// ObjectHandling/GlobalObjects
{attribute 'qualified_only'}
{attribute 'global_init_slot' := '49995'}
VAR_GLOBAL CONSTANT
	MAX_OBJECTS : UINT := 750;
	MAX_CYLINDERS : UINT := 20;
	MAX_MOTORS : UINT := 10;
	MAX_FAULTS : UINT := 300;
	MAX_LOGS : UINT := 100;
	MAX_LOGGABLE : UINT := 500;
	MAX_EXECUTEABLE : UINT := 300;
END_VAR

VAR_GLOBAL
	CollectionOfAllObjects : FB_CollectionHandlerAll; 
	CollectionOfFaults : FB_CollectionHandlerFaults; 
// 	CollectionOfCylinders : FB_CollectionHandlerCylinders;
// 	CollectionOfPositionableMotors : FB_CollectionHandlerPositionableMotors;
	CollectionOfActiveFaults : FB_CollectionHandlerActiveFaults; 
	CollectionOfLogs : FB_CollectionHandlerLogs; 
	CollectionOfLoggable : FB_CollectionHandlerLoggable;
	CollectionOfExecutable : FB_CollectionHandlerExecutable;
	CollectionOfInitialzable : FB_CollectionHandlerInitializable;
	Reversing: INT;
END_VAR

// RemoteComms/RemoteComms
{attribute 'qualified_only'}
VAR_GLOBAL
	OPCInputsToBagger : OPC_Inputs;
	OPCOutputsFromBagger : OPC_Outputs;
	modbusInputsToBagger : Modbus_Inputs;
	modbusOutputsFromBagger : Modbus_Outputs;
END_VAR

// UN00 - Sharp Bagger/UN00_Globals
{attribute 'qualified_only'}
VAR_GLOBAL
	simFaults : FB_Simulation();
END_VAR

VAR_GLOBAL CONSTANT
	sAutomatic : STRING := 'Automatic';
	sSemiAuto : STRING := 'Semi-Auto';
	sMaintenance : STRING := 'Maintenance';
	sSimulation : STRING := 'Simulation';
	
END_VAR

// FBs/FB_CycleCounter
FUNCTION_BLOCK FB_CycleCounter
VAR_INPUT
	reset : BOOL;
END_VAR
VAR_OUTPUT
END_VAR
VAR
    count : UDINT;
END_VAR

IF reset THEN
	THIS^.Clear();
	reset := FALSE;
END_IF

METHOD Clear
VAR_INPUT
END_VAR
count := 0;
END_METHOD

METHOD Increment
VAR_INPUT
END_VAR
count := count + 1;
END_METHOD

METHOD SetCount
VAR_INPUT
	countSetting : UDINT;
END_VAR
count := countSetting;
END_METHOD

END_FUNCTION_BLOCK

// FBs/FB_CylinderLeak
FUNCTION_BLOCK FB_CylinderLeak EXTENDS FB_PredictiveMaint
VAR_INPUT
	iExtended : BOOL;
	iRetracted : BOOL;
	maximumStrokeTime : REAL;
END_VAR
VAR_OUTPUT
	strokeTime : REAL;
END_VAR
VAR
	strokeTimer : TON := (PT := T#1H);
	extendedONS : R_TRIG;
	retractedONS : R_TRIG;
END_VAR

extendedONS(CLK := iExtended);
retractedONS(CLK := iRetracted);

IF extendedONS.Q OR retractedONS.Q THEN
	strokeTime := TO_REAL(strokeTimer.ET) / 1000;
END_IF

strokeTimer(IN := NOT iExtended AND NOT iRetracted);

END_FUNCTION_BLOCK

// FBs/FB_PredictiveMaint
FUNCTION_BLOCK FB_PredictiveMaint EXTENDS FB_CycleCounter
VAR_INPUT
	target : UDINT;
	name : STRING;
	units : STRING := 'Machine Cycles';
END_VAR
VAR_OUTPUT
	
END_VAR
VAR
	
END_VAR

SUPER^();

END_FUNCTION_BLOCK

// FBs/FB_DeviceTreeEnable
{attribute 'analysis' := '-169, -34'}FUNCTION_BLOCK FB_DeviceTreeEnable
VAR_INPUT
	rootEIPNode : DED.INode;
	rootModbusTCPNode : DED.INode;
END_VAR
VAR
	reconfigEIP : DED.Reconfigure;
	reconfigModbusTCP : DED.Reconfigure;
	deviceState : DED.DEVICE_STATE;
	_recongfigCommand : BOOL;
	state : INT;
	disabledSettingWordEIP : DWORD;
	disabledStatusWordEIP : DWORD;
	disabledSettingWordModbusTCP : DWORD;
	disabledStatusWordModbusTCP : DWORD;
END_VAR

VAR_OUTPUT
	
END_VAR

//    Program: FB_EIPCommsConfigure
//    Description: Allows configuration of individual EIP in in the device tree (enable/disable) 
//    For example, to turn off the comms to a Keyence BCV if it isn't installed
//    Created by: Ben Hess
//    Created Date: Wednesday January 6th, 2021

//  Get enable status property
disabledSettingWordEIP.0 := NOT Cube67_BN_E_V2.Enable;
disabledSettingWordEIP.1 := NOT FestoManifold.Enable;
disabledSettingWordEIP.2 := NOT MSFMotor.Enable;
disabledSettingWordEIP.3 := NOT Bag_Delivery_EIP_Motor.Enable;
disabledSettingWordEIP.4 := NOT Bag_Delivery_Rear_Motor.Enable;
disabledSettingWordEIP.5 := NOT Keyence_BCV.Enable;
disabledSettingWordEIP.6 := NOT Infeed_Conveyor_IO.Enable;
disabledSettingWordEIP.7 := NOT Panther_PA.Enable;
disabledSettingWordEIP.8 := NOT IBD_Motor.Enable;
disabledSettingWordEIP.9 := NOT DM374_BCV.Enable;

disabledSettingWordModbusTCP.0 := NOT ModbusTCP_Slave_Device.Enable;

// Get actual enabled state
deviceState := Cube67_BN_E_V2.GetDeviceState();
disabledStatusWordEIP.0 := deviceState = DED.DEVICE_STATE.DISABLED;
deviceState := FestoManifold.GetDeviceState();
disabledStatusWordEIP.1 := deviceState = DED.DEVICE_STATE.DISABLED;
deviceState := MSFMotor.GetDeviceState();
disabledStatusWordEIP.2 := deviceState = DED.DEVICE_STATE.DISABLED;
deviceState := Bag_Delivery_EIP_Motor.GetDeviceState();
disabledStatusWordEIP.3 := deviceState = DED.DEVICE_STATE.DISABLED;
deviceState := Bag_Delivery_Rear_Motor.GetDeviceState();
disabledStatusWordEIP.4 := deviceState = DED.DEVICE_STATE.DISABLED;
deviceState := Keyence_BCV.GetDeviceState();
disabledStatusWordEIP.5 := deviceState = DED.DEVICE_STATE.DISABLED;
deviceState := Infeed_Conveyor_IO.GetDeviceState();
disabledStatusWordEIP.6 := deviceState = DED.DEVICE_STATE.DISABLED;
deviceState := Panther_PA.GetDeviceState();
disabledStatusWordEIP.7 := deviceState = DED.DEVICE_STATE.DISABLED;
deviceState := IBD_Motor.GetDeviceState();
disabledStatusWordEIP.8 := deviceState = DED.DEVICE_STATE.DISABLED;
deviceState := DM374_BCV.GetDeviceState();
disabledStatusWordEIP.9 := deviceState = DED.DEVICE_STATE.DISABLED;

deviceState := ModbusTCP_Slave_Device.GetDeviceState();
disabledStatusWordModbusTCP.0 := deviceState = DED.DEVICE_STATE.DISABLED;

// Compare desired status against state - if different do a reconfigure.
CASE state OF
	0:  reconfigEIP.xExecute := reconfigModbusTCP.xExecute := FALSE;
		IF (disabledSettingWordEIP <> disabledStatusWordEIP) 
		OR (disabledSettingWordModbusTCP <> disabledStatusWordModbusTCP)
		OR _recongfigCommand THEN
			state := 10;
		END_IF
	
	10:	// Set appropriate reconfig - don't want to reset EIP comms if changing Modbus and vice versa
		IF (disabledSettingWordEIP <> disabledStatusWordEIP) OR _recongfigCommand THEN 
			reconfigEIP.xExecute := TRUE;
		END_IF
		IF (disabledSettingWordModbusTCP <> disabledStatusWordModbusTCP) OR _recongfigCommand THEN 
			reconfigModbusTCP.xExecute := TRUE;
		END_IF
		_recongfigCommand := FALSE;
		state := 11;
	
	11:	
		IF (reconfigEIP.xDone OR reconfigModbusTCP.xDone) 
			OR (reconfigEIP.xError OR reconfigModbusTCP.xError) THEN
				state := 0;
		END_IF
END_CASE




reconfigEIP(
	xExecute:= , 
	xDone=> , 
	xBusy=> , 
	xError=> , 
	itfNode:= rootEIPNode, 
	eError=> );

reconfigModbusTCP(
	xExecute:= , 
	xDone=> , 
	xBusy=> , 
	xError=> , 
	itfNode:= rootModbusTCPNode, 
	eError=> );

METHOD ManualReconfig : BOOL
VAR_INPUT
END_VAR
_recongfigCommand := TRUE;
END_METHOD

END_FUNCTION_BLOCK

// FBs/FB_DriveTemp
FUNCTION_BLOCK FB_DriveTemp EXTENDS FB_PredictiveMaint
VAR_INPUT
	iDriveTemp : DINT;
	maxTemp : REAL;
END_VAR
VAR_OUTPUT
	DriveTemp : REAL;
END_VAR
VAR
END_VAR

DriveTemp := TO_REAL(iDriveTemp) / 10.0;

END_FUNCTION_BLOCK

// FBs/FB_FaultHandler
FUNCTION_BLOCK FB_FaultHandler
VAR_INPUT
END_VAR
VAR_OUTPUT
END_VAR
VAR
    faultSourceList : ARRAY[0..100] OF IFault;
    sourcesInList : INT;
END_VAR

METHOD registerFaultSource
VAR_INPUT
     faultSource : REFERENCE TO IFault;
END_VAR
faultSourceList[sourcesInList]:= faultSource;
sourcesInList:= sourcesInList + 1;
END_METHOD

END_FUNCTION_BLOCK

// Interfaces/IFault
INTERFACE IFault EXTENDS IAllObjects

METHOD Ack
VAR_INPUT
END_VAR
END_METHOD

PROPERTY FaultActive : BOOL
END_PROPERTY

PROPERTY FaultID : DINT
END_PROPERTY

METHOD Trigger
VAR_INPUT
END_VAR
END_METHOD

END_INTERFACE

// ObjectHandling/IFault
INTERFACE IFault EXTENDS IAllObjects

METHOD Ack
VAR_INPUT
END_VAR
END_METHOD

METHOD Trigger
VAR_INPUT
END_VAR
END_METHOD

END_INTERFACE

// Interfaces/IAllObjects
INTERFACE IAllObjects EXTENDS __System.IQueryInterface

PROPERTY InstanceName : STRING
END_PROPERTY

END_INTERFACE

// FBs/FB_HMILight
FUNCTION_BLOCK FB_HMILight
VAR_INPUT
END_VAR
VAR_OUTPUT
	lightOutput : BOOL;
END_VAR
VAR
	_turnOn : BOOL;
	_blinkFast : BOOL;
	_blinkSlow : BOOL;
	blinker : OSCAT_BASIC.PWM_DC := (F := 1, DC := 0.5);
	slowBlinkSec : REAL := 1;
	fastBlinkSec : REAL := 0.5;
END_VAR

IF _blinkFast THEN
	blinker.F := fastBlinkSec;
ELSIF _blinkSlow THEN 
	blinker.F := slowBlinkSec;
END_IF
	
blinker(F:= , DC:= , Q=> );

lightOutput := _turnOn OR (blinker.Q AND (_blinkFast OR _blinkSlow));

METHOD BlinkFast
VAR_INPUT
END_VAR
_blinkFast := TRUE;
_blinkSlow := FALSE;
_turnOn := FALSE;
END_METHOD

METHOD BlinkSlow
VAR_INPUT
END_VAR
_blinkFast := FALSE;
_blinkSlow := TRUE;
_turnOn := FALSE;
END_METHOD

METHOD TurnOff
VAR_INPUT
END_VAR
_blinkFast := FALSE;
_blinkSlow := FALSE;
_turnOn := FALSE;
END_METHOD

METHOD TurnOn
VAR_INPUT
END_VAR
_blinkFast := FALSE;
_blinkSlow := FALSE;
_turnOn := TRUE;
END_METHOD

END_FUNCTION_BLOCK

// FBs/FB_TCPClient
FUNCTION_BLOCK FB_TCPClient
VAR_INPUT
END_VAR
VAR_OUTPUT
END_VAR

VAR
    // =======================================
    // set up Client
    // =======================================
    _TCPClient : NBS.TCP_Client;
    _TCPClient_ipAddr: NBS.IP_ADDR;
    _TCPClient_uiPort: UINT := 9100;
    _TCPClient_hClient : CAA.HANDLE; // Client handle
    _sClientIP : STRING(15):='192.168.10.160'; (* this device's Client IP address *)
    _uiPort : UINT:= 9100;
    _TCPConnection : NBS.TCP_Connection; // TCP connection instances
    _TCPConnection_hConnection: CAA.HANDLE;    // handle of client connections    
    _TCPWriteSendLabel : NBS.TCP_Write; // TCP write
	_TCPWriteClearLabel : NBS.TCP_Write; // TCP write
    _TCPRead : NBS.TCP_Read; // TCP read
    _sTCPSendLabel: STRING(25000); // This is the label
	_sTCPClearLabel : STRING(3) := '~JA';
    _sTCPReadData: STRING(1000); //receive up to 1000 chars if needed
    _TCPWriteEn: BOOL;
    _sServerIP: STRING(80);
    _sendLabel : BOOL;
	_clearLabel : BOOL;
	label203 : STRING(8000) := '^XA
^LRY
^LL1218

^GFA,26624,26624,00104,:Z64:
eJztm73u5LYRwCUQiK4IzPYqs/ALGLjGRQAG8IsEyEukOJh6NOVNZLhweUq3gRfLiJwZfkui9iTFOGiK/3+1kvgjOR8kh9ymueWWW2655ZY/g7TtNRx2Eadrh0s4vB0v4Yh2uoQj28clHNU+L+Ho9nUFptWtvoLDZk7/DXH4zBm/IY6cOVc40FUcPXOucFTDucBRmeFcYNjAGU7ncMsZvxmOtJzzDVtZzvmGrS3ndMNugXP6CMSQ05/M6ZAznMzhyBlP5gjknD2FkxdxFHLOdqCLOAZhOSc70FWcznH6izjDqRzhOKFha5SxooS6RcA6p6YIVqVZ5TihYROnZvjjVT2+wamoq6jpXUsATlikdJztMmRNyGpBCymnBYSqCROypnM76DGVGnZnHapqnFXVnAf005hxDL8/hCPAokVq2A1weIWCqoxSQENEZsPA6SrGpSoOKqZLDRt7rGZiV8XREEFZ5vyoGXUMhxynXeLI7dBTYweuHTodGZAjtg27huP0kjmQBA7fHi9q/JSTnanUgZDTHcNxfpM5kIQOY9sOVBNH5SJHOM6WA1VzhsbFn4zTbHNqxh9nZpkDec5W79eMp248WORsW23F/CAoPXUgzzlgpVfBqQgI28K99tMR6HjOROWexwkaETQt4lQEuErOYD+mDkTl8yMm3oHyU8M+ntOczonKTgz7cA6Ny8kIdCQnsjF5MofCcTIyBJwhf3OfRDEgcSDiVAyomxKpJJnCHcmJTCwx7AM5bcRpT+MkLYgd6EBOopHYgY7meAuTZ3FyjwkuD/SfhMPXOGPTwC3XzyxZSCxPR5KIFqsrjjvdOHeruXSGw7wJdRPcWQpQigwMZshshSPM2ruHugx033z6aF6f8O3JtjsVlzTgGH2C0SjhMD3CFoR0lgM2ZOaIzE+c+67Qec4x6eVlTqdHmNArajJmUDp7c2rIWr/rcg7pg5GDRvqKOFKP3HTLXDqD77l+GAuR8/NgPPphWvyx7cucB/435csSRxiOdpxnQ+s808KHsv8m075hruf46decQ2ZtizfAyM6Fm79pU5NRmEc6m2owujRWYds/SvuOUZTQ06fHUOaMlJt6YsNyzst8HpV5RMy15mAzLxq+gMO1eX/64cPfMw5UB81O6yQOhRxNHGmfsjbzRMcmjq3n9M8P/yhzelSPUUzkQClHQ7rJ9NAD/4Qc8TQ6mn7+mHHIfUz3fdFoTd6wiaMgm/Wr5Whb2hMbxfQfZCCNtI2cfn6UOS9boM1XTfEIRBwdcOz2tN3T5aD7/84cSAHZmKBKHHIfhfmDZ+xAnmPMTP9mVNeiOzdgDDNxNmXwHwWcgh0QB1QvvQGlnMko7rfX/BxEGOhs4EibdDRdYWNCiYPe0rp8ROxAIlzXa/377EBT51xH2mbrVzf/F/YJc0dMnz4MKQcr37l1Yx9N4ZDTYfj8Mut7ghU8cPoGNuD7gMOnH/O4g8rgbt04RoYtKI5BRPrSMz0ITJUNMEiYv9/bMNC0yPlrHkfRuLhbN47RBMhzekj2lDlNyOmm7/6yxKGsCScHijnwz3DmLiLOmHEYcrrvUwzVXbr13CNyIOQo5MxPfsBnwZZLHDY1WZKGdKHcOuvpQlHEeRKnsWGHOA32YMQppE7Itkw5tp7qFS3ugcPIu6x1qFfMkQmndOyMk/vY7hobG4tLnCnnTDs4KMZQOMa56AZwBMQhTBlC7+kixypmmcMch8fTL29oCad9i9NZZ4BxaMg4NBmErRcaEWdozrGIzyucvgGlsDj9KDDgPSs5z3UON46uYcqXcWgCaYPSBse2+8dFjni5aUGcCBVYZl/J2Vj9zxyOpcUJSuQAGzjMP5FyNg/MCDNZQm8vcYY1ThhHl/Y7OMSdef6gsDT4GPipi0HbnMYPkGWOemConAt7ggICjs/JVHDKDcJ4rSfXteLJgjaIMI8InG6dU24QlNnQwsa08NXt4PTur+OUE5ygZjv/6pEjcEza5ijkNMSRiw2ynH/roaMCv55TNG175z+GgwrstAoeLnB4wsHThpYTVrHI6Tlx2A6O9dCMU1SQvfOHmVxMxAkiwCZnbCioCVj/BO4WCa5HerdNhJyxhiOA83CcLnx3gTNEnOEtDgv7IhKMvm5iRV/0Kxzn8hzWWZPjgPmWDM5zki++glMMPQpMUTprjB4t+o9PIsF0bPAcscVRMSddB0cc96g1aUUZhqlBgys6ELqWcpWIVLnOaSB7EXCaTU4QHOs50iRCniFHLjlqhxxnjKFZlzgs4EQ7YfBfncYZIo5Y4GBqS430hQpbXuT4rwJtuMClyoEHOT5Y7OCEB5hEEBKHUoMUcIb4epVD9eUmheKeRE63zunj62VOcOpcBpFskyOsW8acLK8cc6icsEDD6fr4fokTta+W0/ubljOscLoCxz1Y5oz28m/RUQDHwfXq/43TWo73vcihCxx3tuIz/1pOvs8UcujMw2ee6Wdc4cCk+JfzOSrj5PuAMQfuP4RO/Ae2MpY40hTs15Qq2XUqcGx725kTjJzbHJ5xfDVLHGwjm+zQRdZZyfmXuwzNeonTNyYtRRw3T1zn2PTAPo55gI/EceuS7rHJ+Snk9KscjmekPGciDuR/lhbdKSeYR6gCp8MzbAMnzjPhlDG25I+7OPZMXu84L+IE+bmCyIQTzFtV3InEsWmnvtOBgixHH8lhNlAJTNXs4PCwc+IfG5U4bgvHZWDM98AxDy8eKYoOZbCUM6Scxikl5wy4k1IUlnD8RepMI8G132Jznw1nfJ/jW0ccSWXzEoeF+o0lLDqcPjfxL06II6ivsGUB52H3zZY5wx4OdxyZcuwml++BRGTA4WGzudbR6mDCqqAtM0yfw3LL7kQZoC8s4/gq8LDZkqKkFRpIgy3xES5fcNMmbxbdh57PP8fLZ+aYysUarM3L3rT5dLboPnEbRGRgThNNuGCRGo/pPvH1F64cSFkLEpqijEeFIgcinNkpbeCSOMF66AhOS2aQclikz0zCH+yqoHuXOLhDQxbMHMe8sdxtUejTNRwGIzdetZ7T6GVrixux4xdaIuDUvtHjpz2/eZaOU1s3z2HL0ekAjt+NWYlOmSjHqe0Dz6n7uRCI3s3xv6wXq/by9Rx6Ur7B2aFTl65S9WbtFnY7dBrt057IIbXsMWs3HvGVkJZx+nc4lHqr5tDkYY9Zu8WErA07fnNC1lfNbd8uT0BzoVC4Hm4TEWAIKxO2AofOm+zgcFj58H06hUXZnt/t4vC96yimxHNC9V1AC5TNzdlIBKyddkTrxq0X9vQBxxNUuzjKzXqrhdaAwx6OeOMdeGXnrzt2dxv1wc6fiatwXlwnfrGxE7Szat3+rm7eOi/9hnreErG7q9+Ua5rjjufccsstt9xyyy233HLLLbfccsstt9xyyy23JPI/RQci9w==:58A1

^FX Border
^FO0,0 ^GB812,1218,2,,1 ^FS

^FX Normal type
^FO80,265^A0,7 ^FD7 px The Quick Brown Fox 0123456789^FS
^FO80,277^A0,14 ^FD14 px The Quick Brown Fox 0123456789^FS
^FO80,295^A0,23 ^FD23 px The Quick Brown Fox 0123456789^FS
^FO80,319^A0,32 ^FD32 px The Quick Brown Fox 0123456789^FS

^FX Vertical type
^FO725,557^A0R,14 ^FD14 px The Quick Brown Fox 0123456789^FS
^FO690,557^A0R,23 ^FD23 pxThe Quick Brown Fox 0123456789^FS

^FX reverse type
^FO80,390^A0,7  ^FD7  px The Quick Brown Fox 0123456789^FS
^FO80,402^A0,14 ^FD14 px The Quick Brown Fox 0123456789^FS
^FO80,420^A0,23 ^FD23 px The Quick Brown Fox 0123456789^FS
^FO80,444^A0,32 ^FD32 px The Quick Brown Fox 0123456789^FS

^FX Reverse Type box
^FO25,360  ^GB760,150, 100,B, 4 ^FS

^FX Circles
^FO 203,636 ^GC50,2 ^FS
^FO 253,636 ^GC50,50 ^FS

^FO 303,636 ^GC50,2 ^FS
^FO 353,636 ^GC50,50 ^FS

^FO 403,636 ^GC50,2 ^FS
^FO 453,636 ^GC50,50 ^FS

^FO 503,636 ^GC50,2 ^FS
^FO 553,636 ^GC50,50 ^FS

^LRN

^FX Box with slashed lines
^FO203,576 ^GB406,50,2^FS

^FO203,576 ^GD50,50,2^FS
^FO253,576 ^GD50,50,2^FS
^FO203,576 ^GD50,50,2,,L^FS
^FO253,576 ^GD50,50,2,,L^FS

^FO353,576 ^GD50,50,2^FS
^FO303,576 ^GD50,50,2^FS
^FO353,576 ^GD50,50,2,,L^FS
^FO303,576 ^GD50,50,2,,L^FS

^FO453,576 ^GD50,50,2^FS
^FO403,576 ^GD50,50,2^FS
^FO453,576 ^GD50,50,2,,L^FS
^FO403,576 ^GD50,50,2,,L^FS

^FO553,576 ^GD50,50,2^FS
^FO503,576 ^GD50,50,2^FS
^FO553,576 ^GD50,50,2,,L^FS
^FO503,576 ^GD50,50,2,,L^FS

^FX Picket Fence Barcodes 
^BY2 ^BC,100 ^FO260,720 ^FD1234567890^FS
^BY3 ^BC,100 ^FO180,860 ^FD1234567890^FS

^FX 2D Barcodes
^FO30,1000^BQN,2,6,M,7^FDQA,http://www.pregis.com^FS
^FO320,1000^BQN,2,6,M,7^FDQA,http://www.pregis.com^FS
^FO610,1000^BQN,2,6,M,7^FDQA,http://www.pregis.com^FS

^FX Ladder barcodes - 
^BY3
^BCB,100 ^FO25,550 ^FD1234567890^FS

^XZ';
	label300 : STRING(8000) := '^XA
^LRY

^FO0,0
^GFA,58368,58368,00152,:Z64:
eJzsnE+u5LYRh0UIsDaBtfUiMK/hRRDmSD6B2cAscowcJQJ8gFxBwSxm6QaySAdoiJFIVrFIFvWHb15Liy4bz22JIj+yij+VSHU3zdve9ra3ve1tb3vb2972tredZz80w9kIrP14Ua6fm/vZCKz9tXmcjcDab83zbATWpvmfC5qYGnM2A2ftzHU7G4Kx7qJc/cw1ng3BmJy5rihgaua6ooDpmeuKAmam5d/LmVi4Lihg7UW5Oss1nI2RWW+5xrMxMpOW63oCpizX9QRMW67rCZixXJcTMHFRrtZxXS7T6TzXcDZIYr3nGs8GSUx6rqsJmPJcVxMw7bmuJmDmmlwCuC6W6bTIdTsbJbIOuYazUSLrkWs8GyUyiVzXEjCFXNcSMH1RLoNcl8p0ROC6lIC1hOt2NgyxjnANZ8MQ6wnXeDYMMUm4riRg6qJcmnBdKdMxhOtCAiYo14UErI24bmfjoHUR13A2DlofcY1n46DJi3KpiOs6mY6OuK4jYCbiygXMEBurWtA1ThAxVy5glKtKRkSVE9qEK2s54qrR3a6qO13CNaxzZae3ra/i6o9xVYSKrOqNTLiyTCfmqui6qpovyjX39HqRD4j6qCNVVVqHOAjIg01+aI/PLV3lfXSfAoem1uI48uc/hcvL1xwBfgIwSqAg7rqqAKuaLS2GTVcMbInzwfXgONdx53c7uDrkUtyE/RSu4L3g0dQEcvUVbYgqLonRDlz5eASutiLw67iIOqBiZBZwKwJf1E5igNElAbNn7vhpOM51fLyI84JLy1zy+ISs4qLBXhawwNUfn5BVXO1Brq5CKGq4qGgFiS1ztRWN1HDRMaJjF1uQ0xqn8HN83aJYLwpY4KrZRdIVXES+kCuvhHDp4wJWwxVpaQSZco3h43CsDVV3Tw2uKwoY4ZLHueTxHETs45Ix18FWKrhiaShmOgSmO85V8fwYk3QRZZnrYLS0x7liiS9mYISrrVCj47IaR1QxAyNcooJLH56OiTJEqlHm+vy1qASkJGAJ1+cvppvDXM0ruNJAL2U6lEsz57+3pZkNcN1O5kqFtJSBvZor9VspA0u5bp/MFctXU8zAKJd6AVc2/woCRrkk4+fvbfqiXJnbMseewpXfpyUvYJSr/3yuXBYKGdiLuXKKQgZGfdczOvKdLb/tFDKwF3MxUc4L2Iu51EW5GLXKlJbl+uS3P5jB4QXstVxckPMZGOWqWWk6ZlxWwwvYa7k4BsGwvpqL8xkvYK/lklwsXYCL1QRGO17NxSKwsK/lYrWdFbCXcvEhzgrYS7n4hzI4eitxfbre8xLK0r6Ui3+4ZoWV5RLj/EdBER1d0BUeffsdSxtshPOzgeXqx+V/HnjVPS4/Upx7uJYeZ41VBF49Ui5btxqXOtzlyX6pTupVd/44axFAhy1zuByXWP7CxFXREPcYCdbXM3XYXHIX/7rCFTks9IRzL8fVzX8FHI+HWGLF/cNdEjYJbTGxsvISyVcfPsI03eLS898OGaNLQs9c96DzCqZUv/KkFwmCDh3m5INy+c8CXgUZsVtQJEigsNW0dHPcDuTPzr+s0fbxnbmGF1aGq12IpIl2oMe4ZvtKxmDPOmHxxx/NX1Z+fIbecODz2PC3J4ZLLSW051q6oTDA5hKj2z9VS1HhCy2UfjPy1+aXIpckY6RwhJvi0whwKffZAJd7n2haWvVzWC+DvZwaDDjbvxTysJc/mq/3MpdneRIUB6lhtNe4bMQLX4H1KWqGsMfABffw8oVcSln836c/FblI8xBSLqgoMMOlbTFJuTrLpXxMtrZSCLJ7i1zKx+XMZX4scpEwksg1NuSFwzKXf7Gp8+WkJZK+jKPEPZ3w0pHjnrnEly8/lLBoeEN4udFjMrCMq424lC3cBS0cQr8jLnf9KhddetbI9WxYYc24bJnRf5FmacpdB+883UKlgUtA+D7bL1+6EheRL2GCNWwGRrlM4JKeC6PUzhU3euCEwNW6kO1nrrYrcvU5SII5slxu3yriEjAermHtxkWmXB3hMkUuf9mEiP9CGIiMItfTx5dyNbS+Dyg6k+/4H7YW7evq4T43c01tiUuFgJLOa9gxHxlEwAiXE3JBuTpMKiYybDPXVwPveTou/2rb6niRxrUJAoGckYARrs5dtDQ2+mLw/rOGMID7/8MStQZuov4uOXOV4544y4cZbnkSFxe5ZJELsodlGujls8i4VnSCbGWHnWHtAHMBS7juPgsz/7OXSl/UcXWB66nsZ8+l/Exa5SJiEFLo5dONy8AIl0+5ls782ycRyg+tguogq3l2kHq4sAWu5vciF2m7w6FpDaRWwJxzycD11bjUinCNFnwELkHzL+2r0AtX6f5IfCWj/e2xtD0zYBH7cf7vt8kNDlwv7SUSii4Rqv2Nk3KpqRmbnwpcJLZlkCoZJoJJt7M8l/YOng99ezrpKnKZ5WfFMq75WDkvVMZPJtuSbxNyO38yCBjhggmxcNm5Ngjy2tEdoszV24gH7S1y/VLMo3VoWkf7yIQrCFjMBbeZP+xcu61xkePI1U8rzx0mcMX7yKyABS4UFc+lDd6GfKAqmMgJlyBc/d8HHouEdksdpngBC1wd4VoOzQ+uCZcmXDeOq1vuqIXhIlLQJgF+YwQscPUQd3Dob5gPHuAq/uYlablP9kUHRsAClzSeQiJ3T849w+NHmE8JV3GwmshT0beOOl7AApeGT9tcqoKLRLakybmIMp07LW4rFeheaUhY3wBkD9faoolyDTtRmLCvkBLrMFtzrgkP4UmsdPogl6ZczybIpbYwBDvm6ijXlHDpLa7Rndj3eo9eLsJcVRluqiCXMuSmM2H7x7j0Li5Mp4y7Z3Ars8ilDRGFZ8zlfbzCBauZe7Cc23WYnWtcHYY9yUJ8TMAE3+ZSzQ4TsDpjYF6ucEljSLQf5vIXqNsOrnapxgvp2PgVvgJXSyZDDRc4fg+XHSAv//cNLgWzAxs7xgUTeAeW4/Ly/1jncvRDymV2c/kTf97D1S+jq1ylLksceS5vUzh0nIupusz1iGR2i+sRDoVvfOzlOrDfJZeWbJWjr425WNKGc65IiktcB78ZIv0TcZj/q1z0lrnBpeP8qyHBWTSNwbI8BbdhuOz4Qf4V3R/jI5VcW9t8Cr2i/HYKTMOecCUbPpEfjnNp0vuSSWxH2+2a0JPOLYRYu6fFhw9zbezy9dgQLHoDQ+sWQshMaKLntENcUVEd+4C1LuJSpNnWbZ/Ew7PG1R7jWo8wiKB743wZiovwjXzueWibC91nEi6VBC1nuLUlPNcznJlQKSnEx7l8dKwPmG/5Kdx6MhEtY2AwueftbS4VHgWmqCjdtCua9k23fhE3FDYGgo9dn/g41+rNSCVcoVVjoAJ2PecI1zMqmlfLmHe2+eIX48MZbf6RdWyNqytwtSlXHh6M9cj1WGomZZX5ZxYIR7ikv7DItfqtAoihbzNXH42tgsv59dVNrj7sGj+ioiKvNzeA/+98SR/FYuAK/arkSlJuqHct8EM2d8cV5MDgLD62lwt4epKiuCN6T+ATLpnt6aXxeZDrwXOBJ1bv3TriujFc/P7QJhfEe+gtFJV7uDCMxrDA0Ph+ZsO9wRXNfNBThb2VIeLSAMlNUi5aMXLx+4/fg+u2woXND8kaTheAd3G1qVJq2PfPHun2cHWU68Gf+AiXYLhUXnNmbWhe81wxxBpX9lLpSOUrFN2TUQjKRZXuw1xOWDmu8g8jEAtccUHgKr1vssnlhEOGWrEoiNMql8YgjNvMHh6PcrkFEhLegcv3eVXw1QZX6X2mTa4FaaBHA1ezg0sSrhs5Hh5J9nEJk058lbROuMQ2V0+46HEuOI9xyaQCwuWYV7kgvpuESyDvfq7onMCKGa4mDd3M2sCV3kc+xtWl8ybiUltc2C3BcyUQ+7lkGp8R10K96xGySX72kL4zupdrzK9/MkXh9DqXXuUqvh+9xTXHx39Metcnk3uTSyFXND88V3RsjatJuPpMzmMubdYTMIiDGSR6EBBpeGxz/R8AAP//7Z1NsqwsDIbbcsDQHVx2ctnZxaWxFJfQQwddx688CCQEEI1VXw/yzk4fSD9iCP80SmxKp/izcU2TK9xTW+ZCGHojjZqGjR4sXPqWfFK1pK9tcqnIhb6SzVW6JWLnendyjU2u+RaXyr2VcqkzrqHJlVtucsUimtyIvYJy0XY+V4uLnrdqccXUk1N8Lhu4HOWi59OqXAZwaVdYlzi41l4u0+DCTnLGlbpaTlf9q5tLB66Zci0kZZVLg1piZl2tj59kv801HQ7+AJeLXIUNBVe5VIPLoZTdXHbfCcnlGhtc6KM2FzzcZffKlKUMXOCypTZXWN6jw5k8pznjiuOK0qVtV7leda6sjWtyqVR9x80Hn7nEtXVz2SpX5rtNLnCl4fgDdwd8UNILXMZz/UMfpnMiF7iO8p0QF573BVxnq6Pal/kDXGGL2gdxofUOdaTp4JqqXBlEkyvtVXtpzIXWRS9wKZ/3L+VyF7he6UHsirlWkFSlnaZnRzPHKtd8lcsTbCuY/o+eH7iWYP+Ma/BFg7nURiuMbXLZ4Ep73wtxbWWu9lryK2xp+EO4cgc459p81iVOxwAHC1xx/ueUy1a48oyWVlHA9VtE75ffQ4O53impOqz2cJlfLrxH/ybXBxwhPeNqLRAF40WuPGObSx+vTKXNWEHrPa7SOe/SZ20ugDKjw1tpReaX6yekzs0TqQqXu8+Ft139pKRXuEb6fahbDLlWkizkHBGGRWCQawvPnT82UWmvmN5oe781uVIRgcMOJa754Mofm6rAZWg8LnV9AFday9zZseM7yOWOjOdctp+LXo0Uc8ZX9369MgejXKZn15yhsarw0SUu7GAL5Fq8/b47KAoxNC9C/2rmKpeGpYMjBeJavf2Oa1Kn4v0Ty0WuCXENVS6ww/9EinJttB6b+BVlrlhCkdKFTG/Itb36wn2xM0RKprzTDboh3uFiDgMmcJl40HzuC6vFTi39ZISlAVjJtZrrYRJMqKz+v5/YtpieMAE2jzVIg1s7nAx8gQHVcYwJj7NGg3+m4yJl27e5liQrdL+D90C/UOjN6uTksb2JJJN/Jr+gQFbDKyLFSrttJlauBByC+oz+nH3ymN+Cn8NJPewOty+0CrS+dHDBOVmL4i3g6trHF0Rad1pfOrjAsuIA8mvEFRekekQwaDekh2uKBTGC/BmXzoy0NBbiZZakhyuFDdiNmTBXaa6npiF3p5tcGgyuY6qc68qv3tA4ntfjLq4BTEbAVIirN6jushlXV3PftJdx3VQ+f5xzXpUF5d0zhK0p96fOuFcTasb6+g5lTWSXwnKf6kEuhV3xxm8hII0Z18Iw5MCf6lu4Bsw1dbYTNamnuDJHL5/L7BfiUh1D66os4iqfY+2X2nD8crctYRJu+EJc936Q8hB+c8zwRbjuW0KZB07J79q5ogXaB7hmaYZ/uGrKTmuQi1GJUADjhi8808eqRKjlYZX8LjTTx6tE+F4M5m+ZjBswx6tEFg2ceeELbTtj9gFMencDo8MULcBxrWOY0in7xOzlxCWnYG1mmAIwfK50W2HnjGVdoBduuOHLj8XivY+sSpS6THTr7nWZOEzi9O4xDWrcbkrHkbfitrU2PJhhh4m06ac4IXpNJrzIjR0mwuTiu2Mf4anCRha98asjusaAWfjh+PbGLvldNnHx3MtPNry9x/K50nQG1xhcCGBjgXUrZhcAFj27OsKnZNch/ZRH/CquysyPWXqgOpYP+txTKvoHsPCsOU8Putcu+5RLhLrN9lSv87MSnQp12z1h7EGVzsB8hfRjUeJZqa98jS9fYN9XXD4Yzv83REn02I9IJBKJRCKRSCQSiUQikUgkEolEIpFIJBKJRCKRSCQSiUQikUgkEolEItG5/gPdo1XZ:DCC5

^FX Border
^FO0,0 ^GB1200,1800,2,,1 ^FS

^FX Normal type
^FO118,391^A0,14 ^FD14 px The Quick Brown Fox 0123456789^FS
^FO118,409^A0,23 ^FD23 px The Quick Brown Fox 0123456789^FS
^FO118,436^A0,32 ^FD32 px The Quick Brown Fox 0123456789^FS
^FO118,471^A0,42 ^FD42 px The Quick Brown Fox^FS

^FX Vertical type
^FO1071,823^A0R,23 ^FD23 px The Quick Brown Fox 0123456789^FS
^FO1020,823^A0R,32 ^FD32 pxThe Quick Brown Fox^FS

^FX reverse type
^FO118,576^A0,14 ^FD14  px The Quick Brown Fox 0123456789^FS
^FO118,594^A0,23 ^FD23 px The Quick Brown Fox 0123456789^FS
^FO118,621^A0,32 ^FD32 px The Quick Brown Fox 0123456789^FS
^FO118,656^A0,42 ^FD42 px The Quick Brown Fox ^FS

^FX Reverse Type box
^FO37,532  ^GB1123,222, 200,B, 4 ^FS

^FX Circles
^FO 300,940 ^GC75,2 ^FS
^FO 374,940 ^GC75,50 ^FS

^FO 448,940 ^GC75,2 ^FS
^FO 522,940 ^GC75,50 ^FS

^FO 596,940 ^GC75,2 ^FS
^FO 669,940 ^GC75,50 ^FS

^FO 743,940 ^GC75,2 ^FS
^FO 817,940 ^GC75,50 ^FS

^LRN

^FX Box with slashed lines
^FO300,851 ^GB600,75,3^FS

^FO300,851 ^GD75,75,3^FS
^FO375,851 ^GD75,75,3^FS
^FO300,851 ^GD75,75,3,,L^FS
^FO375,851 ^GD75,75,3,,L^FS

^FO522,851 ^GD75,75,3^FS
^FO448,851 ^GD75,75,3^FS
^FO522,851 ^GD75,75,3,,L^FS
^FO448,851 ^GD75,75,3,,L^FS

^FO669,851 ^GD75,75,3^FS
^FO596,851 ^GD75,75,3^FS
^FO669,851 ^GD75,75,3,,L^FS
^FO596,851 ^GD75,75,3,,L^FS

^FO817,851 ^GD75,75,3^FS
^FO743,851 ^GD75,75,3^FS
^FO817,851 ^GD75,75,3,,L^FS
^FO743,851 ^GD75,75,3,,L^FS

^FX Picket Fence barcodes 
^BY3 ^BC,148 ^FO384,1064 ^FD1234567890^FS
^BY4 ^BC,148 ^FO310,1271 ^FD1234567890^FS

^FX 2D Barcodes
^FO70,1500^BQN,2,8,M,7^FDQA,http://www.pregis.com^FS
^FO480,1500^BQN,2,8,M,7^FDQA,http://www.pregis.com^FS
^FO910,1500^BQN,2,8,M,7^FDQA,http://www.pregis.com^FS

^FX Ladder barcode 
^BY4
^BCB,148 ^FO37,813 ^FD1234567890^FS

^XZ';
END_VAR

//    Program: PRG_TCP_Client
//    Description: This provides TCP Comms to the zebra printer
//    
//    Created by: Ben Hess
//    Created Date: Tuesday, May 1, 2018

// Here's an example label
CASE HMIData.printerSelection OF
	LabelPrinterSelection.PrintAndApply203DPI:
		_sTCPSendLabel := label203;
		_sClientIP := '192.168.10.165';
	
	LabelPrinterSelection.PrintAndApply300DPI:
		_sTCPSendLabel := label300;
		_sClientIP := '192.168.10.165';
	
	LabelPrinterSelection.ZebraPrinter203DPI:
		_sTCPSendLabel := label203;
		_sClientIP :='192.168.10.160';
	
	LabelPrinterSelection.ZebraPrinter300DPI:
		_sTCPSendLabel := label300;
		_sClientIP :='192.168.10.160';
END_CASE

_TCPClient_ipAddr.sAddr := _sClientIP; // Set IP address
_TCPClient(
	xEnable:= _sendLabel OR _clearLabel, // Manually toggle for testing
	ipAddr:= _TCPClient_ipAddr, 
	uiPort:= _uiPort,
	hConnection=> _TCPConnection_hConnection
);

// set TCP connection
_TCPConnection(
	xEnable:= _TCPClient.xBusy AND NOT(_TCPConnection.xDone), //when server is ready
);

// Write when connection is ready
_TCPWriteSendLabel(
	xExecute:= _sendLabel AND _TCPClient.xActive, // Manually enable for testing
	udiTimeOut:= 600000, // In microseconds => 600ms
	hConnection := _TCPConnection_hConnection,
	szSize := 25000, // Write length only
	pData := ADR(_sTCPSendLabel)
);
// Reset write enable
IF(_TCPWriteSendLabel.xDone) THEN
	_TCPWriteEn:= FALSE;
	_sendLabel := FALSE;
END_IF

// Write when connection is ready
_TCPWriteClearLabel(
	xExecute:= _clearLabel AND _TCPClient.xActive, // Manually enable for testing
	udiTimeOut:= 600000, //in microseconds => 600ms
	hConnection := _TCPConnection_hConnection,
	szSize := 3, // write length only
	pData := ADR(_sTCPClearLabel)
);
// Reset write enable
IF(_TCPWriteClearLabel.xDone) THEN
	_TCPWriteEn:= FALSE;
	_clearLabel := FALSE;
END_IF

METHOD ClearLabel
VAR_INPUT
END_VAR
_clearLabel := TRUE;
END_METHOD

METHOD SendLabel
VAR_INPUT
END_VAR
_sendLabel := TRUE;
END_METHOD

END_FUNCTION_BLOCK

// FBs/FB_Throughput
FUNCTION_BLOCK FB_Throughput
VAR_INPUT
	inCycle : BOOL;
	runtimeTimeout : REAL := 5.0;
	reset : BOOL;
END_VAR
VAR_OUTPUT
	BPM : REAL;
	BPMCycles : UDINT;
	BPMSeconds : UDINT;
	BPMIndication : STRING;
END_VAR
VAR
	resetRuntime : BOOL;
	resetRuntimeTimer : TON := (PT := T#0S);
	runtimeTimeoutTimer : Standard.TON;
	runtimeTimer : Standard.TON;
	actualRuntimeTimer : Standard.TON;
	timeoutONS : FB_ONS;
	inCycleONS : FB_ONS;
	runtimeSeconds : UDINT;
	runtimeMinutes : UDINT;
	runtimeHours : UDINT;
	runtimeDays : UDINT;
	runtimeSubtractedToGetFiveSeconds : UDINT;
	cycleStarted : BOOL;
	totalTempH : UDINT;
	totalTempM : UDINT;
	totalTempS : UDINT;	
END_VAR

// Runtime calculation. The goal is to capture actual runtime of the machine (i.e being used, including loading time)
inCycleONS(CLK := inCycle);
// Reset timeout time 
IF inCycleONS.OSR THEN
	resetRuntime := TRUE;
	cycleStarted := TRUE;
	BPMCycles := BPMCycles + 1;
END_IF;

// After timeout, assume machine in unmanned
runtimeTimeoutTimer(IN := NOT resetRuntime, PT := TO_TIME(runtimeTimeout * 1000.0));
resetRuntime := FALSE;
timeoutONS(CLK := runtimeTimeoutTimer.Q);

// 1 second ticker while being used.
actualRuntimeTimer(IN := cycleStarted AND NOT actualRuntimeTimer.Q AND NOT runtimeTimeoutTimer.Q, PT := T#1S);

IF actualRuntimeTimer.Q THEN
	BPMSeconds := BPMSeconds + 1;
END_IF;

// Subtract 5 seconds after machine is abandoned
runtimeSubtractedToGetFiveSeconds := ANY_TO_UDINT(ABS(5.0 - runtimeTimeout));

IF timeoutONS.OSR THEN
	IF BPMSeconds > runtimeSubtractedToGetFiveSeconds THEN
		BPMSeconds := BPMSeconds - runtimeSubtractedToGetFiveSeconds;
	END_IF;
	cycleStarted := FALSE;
END_IF;

IF reset THEN
	BPMSeconds := 0;
	BPMCycles := 0;
END_IF;


// Concat to string for display
runtimeHours := BPMSeconds / 3600;
runtimeMinutes := (BPMSeconds MOD 3600) / 60;
runtimeSeconds := BPMSeconds MOD 60;

IF BPMSeconds <> 0 THEN
	BPM := ANY_TO_REAL(BPMCycles) / (ANY_TO_REAL(BPMSeconds) / 60.0);
ELSE
	BPM := 0.0;
END_IF;
BPMIndication := '';
BPMIndication := ANY_TO_STRING(runtimeHours);
BPMIndication := INSERT(BPMIndication, 'H  ', LEN(BPMIndication) + 2);
BPMIndication := INSERT(BPMIndication, ANY_TO_STRING(runtimeMinutes), LEN(BPMIndication));
BPMIndication := INSERT(BPMIndication, 'M ', LEN(BPMIndication));
BPMIndication := INSERT(BPMIndication, ANY_TO_STRING(runtimeSeconds), LEN(BPMIndication));
BPMIndication := INSERT(BPMIndication, 'S', LEN(BPMIndication));

END_FUNCTION_BLOCK

// Function Blocks/FB_ONS
FUNCTION_BLOCK FB_ONS
VAR_INPUT
	CLK : BOOL;
END_VAR
VAR_OUTPUT
	OSR : BOOL;
	OSF : BOOL;
END_VAR
VAR
	CLK_OSR : R_TRIG;
	CLK_OSF : F_TRIG;
END_VAR

CLK_OSR(CLK := CLK, Q=> OSR);
CLK_OSF(CLK := CLK, Q=> OSF);

END_FUNCTION_BLOCK

// FBs/FB_WriteToFile
FUNCTION_BLOCK FB_WriteToFile
VAR_INPUT
   xFilePath: STRING;
   xText_Write: STRING(2000);
   xAppend_OverWrite: BOOL;
   xAppend_Pos: UDINT;
   xWrite: BOOL;
   xRead: BOOL;
   xLine_No_To_Read: UDINT;   
END_VAR
VAR_OUTPUT
   xText_Read: STRING(2000);
   xDone: BOOL;
END_VAR
VAR
   
// Write Variables
   xWrite_Trig: R_TRIG;
   xStart_Write: BOOL;
   xNew_Line: STRING(2000);
   
// Read Variables
   xRead_Trig: R_TRIG;
   xStart_Read: BOOL;
   xLine_Read: UDINT;
   
   hFile           : RTS_IEC_HANDLE := RTS_INVALID_HANDLE;
   udiBytesRead    : UDINT;
   udiBytesCopied   : UDINT;
   udiWrite      : UDINT;
   udiFileSize     : UDINT;
   udiPos         : UDINT;

//(* Error Codes *)
   udiPosError          : RTS_IEC_RESULT;
   udiCopyError      : RTS_IEC_RESULT;
   udiDeleteError1      : RTS_IEC_RESULT;
   udiDeleteError2      : RTS_IEC_RESULT;
   udiWriteError1      : RTS_IEC_RESULT;
   udiWriteError2      : RTS_IEC_RESULT;
   udiWriteError3      : RTS_IEC_RESULT;
   udiOpenError1      : RTS_IEC_RESULT;
   udiOpenError2      : RTS_IEC_RESULT;
   udiOpenError3      : RTS_IEC_RESULT;
   udiOpenError4      : RTS_IEC_RESULT;

   udiReadError1   : RTS_IEC_RESULT;
   udiReadError2   : RTS_IEC_RESULT;
   udiReadError3   : RTS_IEC_RESULT;
   udiCloseError1   : RTS_IEC_RESULT;
   udiCloseError2   : RTS_IEC_RESULT;
   udiCloseError3   : RTS_IEC_RESULT;
   udiCloseError4   : RTS_IEC_RESULT;
   udiSizeError : RTS_IEC_RESULT;
   udiDirDeleteError: UDINT; 
   udiCreateError: UDINT;
END_VAR

xWrite_Trig();
//xWrite_Trig.PT:= T#500MS;
xWrite_Trig.CLK:= xWrite;
xStart_Write:= xWrite_Trig.Q;

xRead_Trig();
//xRead_Trig.PT:= T#500MS;
xRead_Trig.CLK:= xRead;
xStart_Read:= xRead_Trig.Q;

IF xStart_Write THEN
   xDone:= FALSE;
   IF xAppend_OverWrite THEN 
   hFile:= SysFileOpen(szFile:= xFilePath, am:= ACCESS_MODE.AM_APPEND, pResult:= ADR(udiOpenError1));
   END_IF
   IF xAppend_OverWrite = FALSE THEN
      hFile:= SysFileOpen(szFile:= xFilePath, am:= ACCESS_MODE.AM_WRITE_PLUS, pResult:= ADR(udiOpenError1));
   END_IF
   udiPosError:= SysFileGetPos(hFile:= hFile, pulPos:= ADR(udiPos));
   IF hFile <> RTS_INVALID_HANDLE THEN
      xNew_Line:= concat('$n', xText_Write);
      IF udiPos = 16#0 THEN
         udiWrite:= SysFileWrite(hFile:= hFile, pbyBuffer:= ADR(xText_Write), ulSize:= INT_TO_UDINT(LEN(xText_Write)), pResult:= ADR(udiWriteError1));
      ELSE
         udiWrite:= SysFileWrite(hFile:= hFile, pbyBuffer:= ADR(xNew_Line), ulSize:= INT_TO_UDINT(LEN(xNew_Line)), pResult:= ADR(udiWriteError1));
      END_IF
      udiCloseError1:= SysFileClose(hFile:= hFile);
   END_IF
   xDone:= TRUE;
END_IF

IF xStart_Read THEN
   xDone:= FALSE;
   hFile:= SysFileOpen(szFile:= xFilePath, am:= ACCESS_MODE.AM_READ, pResult:= ADR(udiOpenError1));
   IF hFile <> RTS_INVALID_HANDLE THEN
      udiBytesRead := SysFileRead(hFile:= hFile, pbyBuffer:= ADR(xText_Read), ulSize:=SIZEOF(xText_Read), pResult:=ADR(udiReadError1));
      xText_Read[udiBytesRead]:= 0;
   END_IF
   //xDone:= TRUE;   
END_IF

END_FUNCTION_BLOCK

// FBs/GetTime
FUNCTION_BLOCK GetTime
VAR_INPUT
END_VAR
VAR_OUTPUT
    currentDateAndTime : DATE_AND_TIME;
    
END_VAR
VAR
    iState                    : INT;
    udiUtcTime             : UDINT;
    udiUtcTimeLocal     : UDINT;
    strTimeDate         : SYSTIMEDATE;
    strTimeDateLocal     : SYSTIMEDATE;
    dtDateTimeUTC        : DATE_AND_TIME;
    timeLeftTime        : TIME;
    timeLeftDWORD        : DWORD;
    dDateUTC            : DATE;
    todTimeOfDayUTC        : TOD;
    
    tSysStartTime        : TIME;
    systimeStartNano    : SYSTIME;
    udiStartTimeResult    : UDINT;
    
    udiResult             : UDINT;
    
    
    GetDateAndTime            : DTU.GetDateAndTime;
    SetTimeZoneInformation    : DTU.SetTimeZoneInformation;
    
    dtCurrent                : DATE_AND_TIME;
    dtConcated                : DATE_AND_TIME;
    eWeekday                 : RTCLK.WEEKDAY;
    uiYear                     : UINT;
    uiMonth                     : UINT;
    uiDay                     : UINT;
    uiHour                     : UINT;
    uiMinute                 : UINT;
    uiSecond                 : UINT;
        
    dtuError                : DTU.ERROR;
END_VAR

CASE iState OF

    0:    
        iState:= 1;
        
    1:  // retrieves the target date and time, including the timezone information which was set before
        GetDateAndTime( xExecute:= TRUE);
        IF GetDateAndTime.xDone THEN
            dtCurrent:= GetDateAndTime.dtDateAndTime;
            GetDateAndTime(xExecute:= FALSE);
			currentDateAndTime := dtCurrent;
            //timeLeft := TIME_TO_DT(DT_TO_TIME(targetDate) - DT_TO_TIME(dttarget));
            iState:= 2;
        END_IF
        IF GetDateAndTime.xError THEN
            GetDateAndTime(xExecute:= FALSE);
            iState:= 32767;
        END_IF
    
    2: (*set a spedific date and time --> returns a variable of type DATE_AND_TIME 
         DateConcat --> set only date information --> returns a variable of type DATE
         TODConcat  --> set only the time information  --> returns a variable of TOD (Time of day) *)
        IF dtuError = 0 THEN
            iState := 3;
        ELSE
            iState := 32767;
        END_IF
        
    3:  (*a DATE_AND_TIME variable is splitted in its parts, like year, month, day etc.
            DateSplit --> the same function for a DATE variable
            TODSplit  --> the same function for a TOD variable *)

            
        IF dtuError = 0 THEN
            iState:= 1;
        ELSE
            iState:= 32767;
        END_IF
        
    32767: ; //error

END_CASE

END_FUNCTION_BLOCK

// FBs/SerialMotorTestFB
FUNCTION_BLOCK SerialMotorTestFB
VAR_INPUT
    runMotorPB : BOOL;
END_VAR
VAR_OUTPUT
END_VAR
VAR
    //testMotor : FB_AppliedMotionStepServoRTU();    
    //orientalMotor : FB_OrientalAZDrive();
END_VAR

(*
orientalMotor(modbusInBuffer := OrientalMotorModbusRead,
                stepsPerInchSetpoint := 2122,
                reversePolarity := FALSE,
                operatingCurrentDefault := 100,
                modbusCommandOutBuffer := OrientalMotorCommandWrites,
                modbusParametersOutBuffer := OrientalMotorParameterWrites,
                triggerCommandWrite => OrientalMotorTriggerCommandWrite,
                triggerParameterWrite => OrientalMotorTriggerParameterWrite);                
orientalMotor.Execute();
*)


IF runMotorPB THEN
    //testMotor.MoveDistance(12,100,100,215);
    //testMotor.HomeNow();
    
    //orientalMotor.MoveDistance(12,10000,10000,10000);
    runMotorPB := FALSE;
END_IF

END_FUNCTION_BLOCK

// Function Blocks/FB_BaseComponent
FUNCTION_BLOCK FB_BaseComponent EXTENDS FB_BaseObject IMPLEMENTS IComponent, IMachineOption
VAR_INPUT
END_VAR
VAR_OUTPUT
END_VAR
VAR
    _ready : BOOL;                    // Ready to be controlled
	_reset : BOOL;
	_makeReady : BOOL;
	_optionActive : BOOL;
	_optionEnabled : BOOL;
	_optionInstalled : BOOL;
	_stateString : STRING := '';
	enableONS : R_TRIG;
	resetONS : R_TRIG;
	makeReadyONS : Standard.R_TRIG;
END_VAR

//	Function Block: BaseComponentFB
//	Description:  Extend this FB for each component as it contains the basic variables and logic that all components must share
//	In all extended FBs must run the parent logic with SUPER^()
//	Created by: Ben Hess
//	Created Date: Friday, June 1, 2018

_optionActive := _optionEnabled AND _optionInstalled;
enableONS(CLK := _optionActive);
resetONS(CLK := _reset);
makeReadyONS(CLK := _makeReady);

METHOD Execute
VAR_INPUT
END_VAR
_optionActive := _optionEnabled AND _optionInstalled;
END_METHOD

METHOD MakeReady : BOOL
VAR_INPUT
END_VAR
_makeReady := TRUE;
END_METHOD

{attribute 'monitoring' := 'variable'}
PROPERTY OptionActive : BOOL
END_PROPERTY

{attribute 'monitoring' := 'variable'}
PROPERTY OptionEnabled : BOOL
END_PROPERTY

{attribute 'monitoring' := 'variable'}
PROPERTY OptionInstalled : BOOL
END_PROPERTY

{attribute 'monitoring' := 'variable'}
PROPERTY Ready : BOOL
END_PROPERTY

METHOD Reset
VAR_INPUT
END_VAR
_reset := TRUE;
END_METHOD

PROPERTY StateString : STRING
END_PROPERTY

METHOD SterilizeVariables : BOOL
VAR_INPUT
END_VAR
//This Method will be used to reset all variables to what they should be in the idle state.  should be called whenever we want to make sure all variables are in a known condition.
END_METHOD

END_FUNCTION_BLOCK

// FBs/Components/FB_BaseComponent
FUNCTION_BLOCK FB_BaseComponent IMPLEMENTS IComponentStatus
VAR_INPUT
	enable : BOOL;                    // Enable
END_VAR
VAR_OUTPUT
END_VAR
VAR
	_mode : DEVICE_MODES;            // Auto-SemiAuto-Manual
    _ready : BOOL;                    // Ready to be controlled
	_reset : BOOL;
	enableONS : R_TRIG;
	resetONS : R_TRIG;
	autoModeSelected : BOOL;
    semiAutoModeSelected : BOOL;
    manualModeSelected : BOOL;
END_VAR

//	Function Block: BaseComponentFB
//	Description:  Extend this FB for each component as it contains the basic variables and logic that all components must share
//	In all extended FBs you must run the parent logic with SUPER^()
//	Created by: Ben Hess
//	Created Date: Friday, June 1, 2018


enableONS(CLK := enable);
resetONS(CLK := _reset);

autoModeSelected := (_mode = DEVICE_MODES.Auto);
semiAutoModeSelected := (_mode = DEVICE_MODES.SemiAuto);
manualModeSelected := (_mode = DEVICE_MODES.Manual);
IF _reset THEN
	_reset := FALSE;
END_IF

END_FUNCTION_BLOCK

// Interfaces/IComponentStatus
INTERFACE IComponentStatus

PROPERTY Mode : DEVICE_MODES
END_PROPERTY

PROPERTY Ready : BOOL
END_PROPERTY

END_INTERFACE

// Function Blocks/FB_BaseObject
FUNCTION_BLOCK FB_BaseObject IMPLEMENTS IAllObjects, ILoggable
VAR_INPUT
END_VAR
VAR_OUTPUT
END_VAR
VAR
	_instanceName : STRING;			// Instance Name
	_prefix : STRING;
	_logger : IMachineLogger;
END_VAR

METHOD FB_Init : BOOL
VAR_INPUT
  bInitRetains : BOOL; // TRUE: the retain variables are initialized (reset warm / reset cold)
  bInCopyCode : BOOL;  // TRUE: the instance will be copied to the copy code afterward (online change)
  name : STRING;
END_VAR
_instanceName := name;
_prefix := CONCAT(name, ' ');
GlobalObjects.CollectionOfAllObjects.AddObject(THIS^);
END_METHOD

{attribute 'monitoring' := 'variable'}
PROPERTY InstanceName : STRING
END_PROPERTY

METHOD RegisterLogger
VAR_INPUT
	internalLogger : IMachineLogger;
END_VAR
_logger := internalLogger;
END_METHOD

END_FUNCTION_BLOCK

// Interfaces/ILoggable
INTERFACE ILoggable EXTENDS IAllObjects

METHOD RegisterLogger
VAR_INPUT
	internalLogger : IMachineLogger;
END_VAR
END_METHOD

END_INTERFACE

// Interfaces/IMachineLogger
INTERFACE IMachineLogger EXTENDS IAllObjects

METHOD AddLogItem
VAR_INPUT
	message : STRING;
END_VAR
END_METHOD

END_INTERFACE

// Interfaces/IComponent
INTERFACE  IComponent EXTENDS IMachineOption

METHOD MakeReady : BOOL
VAR_INPUT
END_VAR
END_METHOD

PROPERTY Ready : BOOL
END_PROPERTY

METHOD Reset
VAR_INPUT
END_VAR
END_METHOD

PROPERTY StateString : String
END_PROPERTY

METHOD SterilizeVariables : BOOL
VAR_INPUT
END_VAR
END_METHOD

END_INTERFACE

// Interfaces/IMachineOption
INTERFACE IMachineOption EXTENDS IAllObjects

PROPERTY OptionActive : BOOL
END_PROPERTY

PROPERTY OptionEnabled : BOOL
END_PROPERTY

PROPERTY OptionInstalled : BOOL
END_PROPERTY

END_INTERFACE

// Function Blocks/FB_Delay
FUNCTION_BLOCK FB_Delay IMPLEMENTS IExecuteAutomatically
VAR_INPUT
	in : BOOL;
	delay : TIME;
END_VAR
VAR_OUTPUT
	Q : BOOL;
END_VAR
VAR
	delayTimer : TON;
END_VAR

METHOD Execute
delayTimer(IN := in, PT := delay, Q => Q);
END_METHOD

END_FUNCTION_BLOCK

// Interfaces/IExecuteAutomatically
INTERFACE IExecuteAutomatically EXTENDS IAllObjects

METHOD Execute
VAR_INPUT
END_VAR
END_METHOD

END_INTERFACE

// Function Blocks/FB_GetTime
FUNCTION_BLOCK FB_GetTime
VAR_INPUT
END_VAR
VAR_OUTPUT
    currentDateAndTime : DATE_AND_TIME;
END_VAR
VAR
    iState : INT;
    udiUtcTime : UDINT;
    udiUtcTimeLocal : UDINT;
    strTimeDate : SYSTIMEDATE;
    strTimeDateLocal : SYSTIMEDATE;
    dtDateTimeUTC : DATE_AND_TIME;
    timeLeftTime : TIME;
    timeLeftDWORD : DWORD;
    dDateUTC : DATE;
    todTimeOfDayUTC : TOD;
    
    tSysStartTime : TIME;
    systimeStartNano : SYSTIME;
    udiStartTimeResult : UDINT;
    udiResult : UDINT;
    
    GetDateAndTime : DTU.GetDateAndTime;
    SetTimeZoneInformation : DTU.SetTimeZoneInformation;
    
    dtCurrent : DATE_AND_TIME;
    dtConcated : DATE_AND_TIME;
    //eWeekday                 : RTCLK.WEEKDAY;
    uiYear : UINT;
    uiMonth : UINT;
    uiDay : UINT;
    uiHour : UINT;
    uiMinute : UINT;
    uiSecond : UINT;
        
    dtuError : DTU.ERROR;
END_VAR

CASE iState OF

    0:    
        iState:= 1;
        
    1:  // retrieves the target date and time, including the timezone information which was set before
        GetDateAndTime( xExecute:= TRUE);
        IF GetDateAndTime.xDone THEN
            dtCurrent:= GetDateAndTime.dtDateAndTime;
            GetDateAndTime(xExecute:= FALSE);
			currentDateAndTime := dtCurrent;
            //timeLeft := TIME_TO_DT(DT_TO_TIME(targetDate) - DT_TO_TIME(dttarget));
            iState:= 2;
        END_IF
        IF GetDateAndTime.xError THEN
            GetDateAndTime(xExecute:= FALSE);
            iState:= 32767;
        END_IF
    
    2: (*set a spedific date and time --> returns a variable of type DATE_AND_TIME 
         DateConcat --> set only date information --> returns a variable of type DATE
         TODConcat  --> set only the time information  --> returns a variable of TOD (Time of day) *)
        IF dtuError = 0 THEN
            iState := 3;
        ELSE
            iState := 32767;
        END_IF
        
    3:  (*a DATE_AND_TIME variable is splitted in its parts, like year, month, day etc.
            DateSplit --> the same function for a DATE variable
            TODSplit  --> the same function for a TOD variable *)

            
        IF dtuError = 0 THEN
            iState:= 1;
        ELSE
            iState:= 32767;
        END_IF
        
    32767: ; //error

END_CASE

END_FUNCTION_BLOCK

// Function Blocks/FB_HMIData
{attribute 'FBVisuCreator'}
FUNCTION_BLOCK FB_HMIData
VAR_INPUT
	initiateCycle : BOOL;  // Initiate Cycle Pushbutton
	ackAllFaults : BOOL; // Acknowledge All Faults from HMI
	makeReady : BOOL;
	pressureBarService : ServiceCommands;
	loadPlateService : ServiceCommands;
    stopMachine : BOOL;
	{attribute 'FBVisuCreatorFormatString' := '%s'}
	version : STRING := '0.2A';
	inCycle : BOOL;
	batchEnable : BOOL;
	{attribute 'FBVisuCreatorFormatString' := '%d'}
	batchSetting : UDINT := 10;
	{attribute 'FBVisuCreatorFormatString' := '%d'}
	batchCount : UDINT;
	{attribute 'FBVisuCreatorFormatString' := '%d'}
	headCycleCount : UDINT;
	{attribute 'FBVisuCreatorFormatString' := '%1.2f'}
	pressureBarOpenDelay : REAL;
	{attribute 'FBVisuCreatorFormatString' := '%1.2f'}
	pressureBarCloseDelay : REAL;
	{attribute 'FBVisuCreatorFormatString' := '%1.2f'}
	passthroughSetting : REAL := 8.0;
	{attribute 'FBVisuCreatorFormatString' := '%1.2f'}
	passthroughActual : REAL;
	{attribute 'FBVisuCreatorFormatString' := '%1.2f'}
	lpaDwell : REAL;
	{attribute 'FBVisuCreatorFormatString' := '%1.2f'}
	hpaDwell : REAL;
	{attribute 'FBVisuCreatorFormatString' := '%1.2f'}
	sealBarDwell : REAL := 0.750;
	{attribute 'FBVisuCreatorFormatString' := '%d'}
	sealBarTemperatureSetting : UDINT;
	{attribute 'FBVisuCreatorFormatString' := '%d'}
	sealBarTemperature : UDINT;
	{attribute 'FBVisuCreatorFormatString' := '%1.2f'}
	sealFlattenerBagOpenPositionSetting : REAL;
	{attribute 'FBVisuCreatorFormatString' := '%1.2f'}
	sealFlattenerFlattenedPositionSetting : REAL;
	{attribute 'FBVisuCreatorFormatString' := '%1.2f'}
	sealFlattenerMoveInPositionSetting : REAL;
	{attribute 'FBVisuCreatorFormatString' := '%1.2f'}
	bagSkirtLength : REAL := 1.35;
	{attribute 'FBVisuCreatorFormatString' := '%1.2f'}
	bagLength : REAL := 23.5;
	{attribute 'FBVisuCreatorFormatString' := '%1.2f'}
	bagWidth : REAL := 17.5;
	{attribute 'FBVisuCreatorFormatString' := '%1.2f'}
	bagThickness : REAL := 2.5;
	{attribute 'FBVisuCreatorFormatString' := '%d'}
	bagForwardSpeed : UDINT := 55;
	{attribute 'FBVisuCreatorFormatString' := '%d'}
	bagReverseSpeed : UDINT := 3;
	{attribute 'FBVisuCreatorFormatString' := '%d'}
	printSpeed : UDINT := 6;
	{attribute 'FBVisuCreatorFormatString' := '%1.2f'}
	printLength : REAL := 8.0;
	{attribute 'FBVisuCreatorFormatString' := '%1.2f'}
	printOffset : REAL := 2.0;
	{attribute 'FBVisuCreatorFormatString' := '%d'}
	fillerCountSetting : UDINT;
	{attribute 'FBVisuCreatorFormatString' := '%d'}
	fillerCurrentCount : UDINT;
	{attribute 'FBVisuCreatorFormatString' := '%1.2f'}
	fillerDropTime : REAL;
	{attribute 'FBVisuCreatorFormatString' := '%1.2f'}
	loadPlateDelay : REAL;
	{attribute 'FBVisuCreatorFormatString' := '%1.2f'}
	loadPlateDwell : REAL := 2.5;
	exitConveyorService: ServiceCommands;
	{attribute 'FBVisuCreatorFormatString' := '%1.2f'}
	exitConveyorDwell : REAL := 9.0;
	{attribute 'FBVisuCreatorFormatString' := '%1.2f'}
	lastCycleTime : REAL;
	{attribute 'FBVisuCreatorFormatString' := '%1.2f'}
	bagDropClearanceDwell : REAL := 0.5;
	{attribute 'FBVisuCreatorFormatString' := '%1.2f'}
	averageCycleTime : REAL;
	resetAverageCycleTime : BOOL;
	{attribute 'FBVisuCreatorFormatString' := '%d'}
	bagOpenRetrySetting : UINT := 3;
	{attribute 'FBVisuCreatorFormatString' := '%d'}
	bagOpenRetryCount : UINT;
	{attribute 'FBVisuCreatorFormatString' := '%d'}
	currentJobID : INT;
	separateBeforeSeal : BOOL := TRUE;
	activateDemoMode : BOOL;
	bagOpenAssistEnable : BOOL := TRUE;
	bagOpenSensorEnable : BOOL := TRUE;
	{attribute 'FBVisuCreatorFormatString' := '%1.2f'}
	grabBagDelay : REAL := 0.5;
	{attribute 'FBVisuCreatorFormatString' := '%1.2f'}
	checkForBagOpenDelay : REAL := 1.0;
	{attribute 'FBVisuCreatorFormatString' := '%1.2f'}
	bagClearedFromFingersDelay : REAL := 0.5;
	{attribute 'FBVisuCreatorFormatString' := '%1.2f'}
	vacuumDwell : REAL := 0.5;
	(*Faults*)
	{attribute 'FBVisuCreatorFormatString' := '%s'}
	pressureBarState : STRING;
    stationValveSelection : ARRAY[1..16] OF ValveSelection := 	[ValveSelection.PressureBar,
																ValveSelection.PressureBar,
																ValveSelection.SealBar,
																ValveSelection.HPA_LPA,
																ValveSelection.LoadPlate,
																ValveSelection.BagOpenFingers,
																ValveSelection.PrintHead,
																ValveSelection.Vacuum,
																ValveSelection.SealFlattenersVerticalAxis,
																ValveSelection.LoadShelf,
																6(ValveSelection.Blank)];
    (*Counters*)
    //baggerCycles : FB_MachineCounter(name := 'Bagger Cycle Counter');
	pressureBarCycles : FB_MachineCounter(name := 'Pressure Bar Cycle Counter');
	//passthroughChanges : FB_MachineCounter(name := 'Passthrough Changes Counter');
	//loadPlateCycles : FB_MachineCounter(name := 'Load Plate Cycle Counter');
	//printerCycles : FB_MachineCounter(name := 'Printer Cycle Counter');
	//motorizedSealFlattenerCycles : FB_MachineCounter(name := 'Motorized Seal Flattener Cycles');
	//bagOpenRetryTotal : FB_MachineCounter(name := 'Bag Open Retry Totals');
	(*Info*)
	faultActive : BOOL;
	simulateAllIO : BOOL;
	
	(*Factoy Config*)
	bofSelection : BagOpenFingersSelection := BagOpenFingersSelection.PneumaticWithBagOpenSensors;
	bofEnable : BOOL := TRUE;
	sealFlattenersSelection : SealFlattenerSelection := SealFlattenerSelection.MotorizedSealFlatteners;
	sealFlattenersEnable : BOOL := TRUE;
	printerSelection : LabelPrinterSelection := LabelPrinterSelection.ZebraPrinter;
	printerEnable : BOOL := TRUE;
	integratedExitConveyorSelection : IntegratedConveyorSelection := IntegratedConveyorSelection.RearExit;
	integratedExitConveyorEnable : BOOL := TRUE;
	packageEjectSelection : PackageEjectionSelection := PackageEjectionSelection.RearRetractingLoadPlate;
	packageEjectEnable : BOOL := TRUE;
END_VAR
VAR_OUTPUT
END_VAR
VAR
END_VAR

END_FUNCTION_BLOCK

// Function Blocks/FB_MachineCounter/FB_MachineCounter
FUNCTION_BLOCK FINAL FB_MachineCounter EXTENDS FB_BaseObject IMPLEMENTS ICounter
VAR_INPUT
END_VAR
VAR_OUTPUT
	count : UDINT;
END_VAR
VAR   
END_VAR

END_FUNCTION_BLOCK

// Interfaces/ICounter
INTERFACE ICounter EXTENDS IAllObjects

METHOD Increment
VAR_INPUT
END_VAR
END_METHOD

END_INTERFACE

// Function Blocks/FB_InternalLogger_1
FUNCTION_BLOCK FB_InternalLogger_1 IMPLEMENTS IMachineLogger
VAR_INPUT
END_VAR
VAR_OUTPUT
END_VAR
VAR
	//loggedItems : ARRAY[0..500] OF FaultLogType;
	loggedItems : ARRAY[0..Globals.MAX_LOGGED_ITEMS] OF LogMessageType;
	numOfLogEntries : UINT;
	logFull : BOOL;
	RTC : FB_GetTime();
	clearLog : BOOL;
	i : UINT;
END_VAR

//	Function Block: FB_Logger
//	Description: This is an internal logger for reference within Codesys.  It is an array that can be displayed on the TargetVisu/WebVisu 
//	
//	Created by: Ben Hess
//	Created Date: Tuesday, September 11, 2018

RTC();

IF clearLog THEN
	FOR i := 0 TO Globals.MAX_LOGGED_ITEMS BY 1 DO
		loggedItems[i].logMessage := '';
		loggedItems[i].logTime := DT#1970-1-1-1:0:0;
	END_FOR
	numOfLogEntries := 0;
	logFull := FALSE;
	clearLog := FALSE;
END_IF

METHOD AddLogItem
VAR_INPUT
	//category : STRING;
	message : STRING;
END_VAR
FOR i := GlobalData.MAX_LOGGED_ITEMS -1 TO 1 BY -1 DO
		loggedItems[i] := loggedItems[i-1];
END_FOR
//loggedItems[0].logCategory := category;
loggedItems[0].logMessage := message;
loggedItems[0].logTime := RTC.currentDateAndTime;
END_METHOD

PROPERTY InstanceName : STRING
END_PROPERTY

END_FUNCTION_BLOCK

// Function Blocks/FB_InternalLogger
FUNCTION_BLOCK FB_InternalLogger IMPLEMENTS IMachineLogger
VAR_INPUT
END_VAR
VAR_OUTPUT
END_VAR
VAR
	//loggedItems : ARRAY[0..500] OF FaultLogType;
	loggedItems : ARRAY[0..GlobalData.MAX_LOGGED_ITEMS] OF LogMessageType;
	numOfLogEntries : UINT;
	logFull : BOOL;
	RTC : FB_GetTime();
	clearLog : BOOL;
	i : UINT;
END_VAR

//	Function Block: FB_Logger
//	Description: This is an internal logger for reference within Codesys.  It is an array that can be displayed on the TargetVisu/WebVisu 
//	
//	Created by: Ben Hess
//	Created Date: Tuesday, September 11, 2018

// DISABLED LOGGING FOR CREVIS PLC - SCAN TIMES OUT OF CONTROL

METHOD AddLogItem
VAR_INPUT
	//category : STRING;
	message : STRING;
END_VAR
END_METHOD

END_FUNCTION_BLOCK

// Function Blocks/FB_LoggableBool
FUNCTION_BLOCK FB_LoggableBool EXTENDS FB_BaseObject IMPLEMENTS ILoggable
VAR_INPUT
	in : BOOL;
END_VAR
VAR_OUTPUT
	Q : BOOL;
END_VAR
VAR
END_VAR

END_FUNCTION_BLOCK

// Function Blocks/FB_MetricConversions
FUNCTION_BLOCK e
VAR_INPUT
    bagLengthIn : REAL;
    bagWidthIn : REAL;
    bagSkirtLengthIn : REAL;
    sealBarTempIn : REAL;
    printSpeedIn : UDINT;
    printOffsetIn : REAL;
    printLengthIn : REAL;
    passthroughSettingIn : REAL;
    jawClosePositionSettingIn : REAL;
    barcodeStartPositionIn : REAL;
    barcodeScanningDistanceIn : REAL;
	feedSpeedIn : REAL;
    reverseSpeedIn : REAL;
END_VAR
VAR_OUTPUT
    bagLengthOut : REAL;
    bagWidthOut : REAL;
    bagSkirtLengthOut : REAL;
    sealBarTempOut : REAL;
    printSpeedOut : UDINT;
    printOffsetOut : REAL;
    printLengthOut : REAL;
    passthroughSettingOut : REAL;
    jawClosePositionSettingOut : REAL;
    barcodeStartPositionOut : REAL;
    barcodeScanningDistanceOut : REAL;
   	feedSpeedOut : REAL;
    reverseSpeedOut : REAL;
END_VAR
VAR 
    _ConvertMetricToInch: F_TRIG;
    _ConvertInchToMetric: R_TRIG;
END_VAR

//    Function Block: FB_ModbusDWORD
//    Description: Automatically converts inches to mm every time an inch value changes.
//    
//    Created by: Steve Olson
//    Created Date: Friday, January 3, 2025

_ConvertInchToMetric(CLK := HMIData.HMIMetric);
_ConvertMetricToInch(CLK := HMIData.HMIMetric);

IF HMIData.HMIMetric THEN
    bagLengthOut := bagLengthIn / 25.4;
    bagWidthOut := bagWidthIn / 25.4;
    bagSkirtLengthOut := bagSkirtLengthIn / 25.4;
    printSpeedOut := LREAL_TO_UDINT(printSpeedIn / 25.4);
    printOffsetOut := printOffsetIn / 25.4;
    printLengthOut := printLengthIn / 25.4;
    passthroughSettingOut := passthroughSettingIn / 25.4;
    jawClosePositionSettingOut := jawClosePositionSettingIn / 25.4;
    barcodeStartPositionOut := barcodeStartPositionIn / 25.4;
    sealBarTempOut := (sealBarTempIn - 32) * 5 / 9; // Fahrenheit to Celsius
    feedSpeedOut := (feedSpeedIn / 25.4);
    reverseSpeedOut := (reverseSpeedIn / 25.4);
ELSE
    bagLengthOut := bagLengthIn;
    bagWidthOut := bagWidthIn;
    bagSkirtLengthOut := bagSkirtLengthIn;
    printSpeedOut := printSpeedIn;
    printOffsetOut := printOffsetIn;
    printLengthOut := printLengthIn;
    passthroughSettingOut := passthroughSettingIn;
    jawClosePositionSettingOut := jawClosePositionSettingIn;
    barcodeStartPositionOut := barcodeStartPositionIn;
    sealBarTempOut := sealBarTempIn;
    feedSpeedOut := feedSpeedIn;
    reverseSpeedOut := reverseSpeedIn;
END_IF

HMIData.HMIMetric; // testing visibility

IF _ConvertInchToMetric.Q THEN
    HMIData.bagLength := bagLengthIn * 25.4;
    HMIData.bagSkirtLength := bagSkirtLengthIn * 25.4;
    HMIData.printOffset := printOffsetIn * 25.4;
    HMIData.printLength := printLengthIn * 25.4;
    HMIData.passthroughSetting := passthroughSettingIn * 25.4;
    HMIData.jawClosePositionSetting := jawClosePositionSettingIn * 25.4;
    HMIData.barcodeStartPosition := barcodeStartPositionIn * 25.4;
	HMIData.printSpeed := REAL_TO_UINT(printSpeedIn * 25.4);
    //sealBarTempOut := (sealBarTempIn - 32) * 5 / 9; // Fahrenheit to Celsius
    HMIData.bagForwardSpeed := REAL_TO_UDINT(feedSpeedIn * 25.4);
    HMIData.bagReverseSpeed := REAL_TO_UDINT(reverseSpeedIn * 25.4);
END_IF

IF _ConvertMetricToInch.Q THEN
    HMIData.bagLength := bagLengthIn / 25.4;
    HMIData.bagSkirtLength := bagSkirtLengthIn / 25.4;
    HMIData.printOffset := printOffsetIn / 25.4;
    HMIData.printLength := printLengthIn / 25.4;
    HMIData.passthroughSetting := passthroughSettingIn / 25.4;
    HMIData.jawClosePositionSetting := jawClosePositionSettingIn / 25.4;
    HMIData.barcodeStartPosition := barcodeStartPositionIn / 25.4;
	HMIData.printSpeed := REAL_TO_UINT(printSpeedIn / 25.4);
    sealBarTempOut := (sealBarTempIn * 9 / 5) + 32; // Celsius to Fahrenheit
    HMIData.bagForwardSpeed := REAL_TO_UDINT(feedSpeedIn / 25.4);
    HMIData.bagReverseSpeed := REAL_TO_UDINT(reverseSpeedIn / 25.4);
END_IF

END_FUNCTION_BLOCK

// FBs/DataHandlers/FB_ModbusDWORD
FUNCTION_BLOCK FB_ModbusDWORD
VAR_INPUT
END_VAR
VAR_OUTPUT
END_VAR
VAR
    _highWord : WORD;
    _lowWord : WORD;
    _rawValue : DWORD;
END_VAR

//    Function Block: FB_ModbusDWORD
//    Description: Automatically handles the packing and unpacking of Upper and Lower words to create a DWORD
//    for 16 bit modbus communications
//    
//    Created by: Ben Hess
//    Created Date: Wednesday, April 11, 2018

END_FUNCTION_BLOCK

// Function Blocks/FB_SimulatedFeedback
FUNCTION_BLOCK FB_SimulatedFeedback EXTENDS FB_BaseObject
VAR_INPUT
	in : BOOL;			// Start of feedback (usually an output)
	simFeedbackFault : BOOL;	// Enable a feedback fault
	faultDelay : DINT;			// Delay for feedback fault
	minDelay : DINT;	//Minimum delay in mS
	maxDelay : DINT;	//Maximum delay in mS
END_VAR
VAR_OUTPUT
	Q : BOOL;
	fault : BOOL;
END_VAR
VAR
	inONS : FB_ONS();
	QONS : FB_ONS();
	_beginTimer : BOOL;
	randomDelay : DINT;
	delayTimer : Standard.TON;
END_VAR

//	Function Block: FB_SimulatedFeedback
//	Description: Meant to simulate a feedback based off an input with an additional option to simulate a failed feedback signal
//				 Can be used for testing or for creating "feedback" for components that lack a sensor
//
//	Usage: simPbarInFB(in := movePbarInOutput, minDelay := 100, maxDelay := 200);
// 
//	Created by: Ben Hess
//	Created Date: 3-2019

inONS(CLK := in);
QONS(CLK := Q);
IF minDelay < 0 THEN
	minDelay := 0;
END_IF
IF inONS.OSR THEN
	_logger.AddLogItem(CONCAT(_prefix,'Started'));
	// Feeback can be set as a range to simulate variations in air pressure, friction etc.
	// Choose a random delay in between min and max
	IF NOT simFeedbackFault THEN
		randomDelay := 	FN_RandomDINT(last := randomDelay,
								low := minDelay,
								high := maxDelay);
		delayTimer.PT := DINT_TO_TIME(randomDelay);	
	ELSE 
		// Use fault timer if fault sim enabled
		delayTimer.PT := DINT_TO_TIME(faultDelay);
	END_IF
END_IF

IF QONS.OSR AND NOT simFeedbackFault THEN
	_logger.AddLogItem(CONCAT(_prefix,'Done'));
END_IF
				
delayTimer(IN := in);

IF NOT simFeedbackFault THEN
	Q := delayTimer.Q;
	fault := FALSE;
ELSE 
	Q := FALSE;
	fault := delayTimer.Q;
END_IF

END_FUNCTION_BLOCK

// Function Blocks/FN_RandomDINT
FUNCTION FN_RandomDINT : DINT
VAR_INPUT
	last : DINT;
	low : DINT;
	high : DINT;
END_VAR
VAR
END_VAR

FN_RandomDINT := TO_DINT(OSCAT_BASIC.RDM(OSCAT_BASIC.FRACT(TO_REAL(last) * OSCAT_BASIC.Globale_Variablen.MATH.PI)) * (TO_REAL(high) - TO_REAL(low) + 1)) + low;

END_FUNCTION

// Function Blocks/FB_SimulatedFeedbackPhysicalInput
FUNCTION_BLOCK FB_SimulatedFeedbackPhysicalInput EXTENDS FB_SimulatedFeedback
VAR_INPUT
	inputToSimulate : REFERENCE TO FB_PhysicalDigitalInput;					
END_VAR
VAR_OUTPUT
END_VAR
VAR
END_VAR

//	Function Block: FB_SimulatedFeedbackPhysicalInput
//	Description: Meant to simulate a feedback based off an input with an additional option to simulate a failed feedback signal
//				 Using a physical input to simulate
//
//	Usage: simPbarInFB(in := movePbarInOutput, minDelay := 100, maxDelay := 200);
// 
//	Created by: Ben Hess
//	Created Date: 5-20-2019

SUPER^();

IF inputToSimulate.simulate = TRUE THEN
	inputToSimulate.simValue := Q;
END_IF

END_FUNCTION_BLOCK

// Function Blocks/IO/FB_PhysicalDigitalInput
FUNCTION_BLOCK FB_PhysicalDigitalInput EXTENDS FB_BaseObject IMPLEMENTS IExecuteAutomatically
VAR_INPUT
	in : REFERENCE TO BOOL;
	simulate : BOOL;
	simValue : BOOL;
	debounceEnable : BOOL;	// 
	debounceTime : REAL := 50.0;		// Debounce time in MS
END_VAR
VAR_OUTPUT
	Active : BOOL;
	OSR : BOOL;
	OSF : BOOL;
END_VAR
VAR
	debounceTimer : TON;
	inputONS : FB_ONS();
END_VAR

END_FUNCTION_BLOCK

// Interfaces/IFaultHandler
INTERFACE IFaultHandler

METHOD AddActiveFault
VAR_INPUT
END_VAR
END_METHOD

METHOD RemoveActiveFault
VAR_INPUT
END_VAR
END_METHOD

END_INTERFACE

// Interfaces/ISupervisor
INTERFACE ISupervisor

METHOD MakeReady
VAR_INPUT
END_VAR
END_METHOD

METHOD NotifyMachineFaulted
VAR_INPUT
END_VAR
END_METHOD

END_INTERFACE

// Interfaces/ICylinder
INTERFACE ICylinder EXTENDS IAllObjects

METHOD Extend
VAR_INPUT
END_VAR
END_METHOD

PROPERTY ExtendAsserted : BOOL
END_PROPERTY

PROPERTY IsExtended : BOOL
END_PROPERTY

PROPERTY IsRetracted : BOOL
END_PROPERTY

METHOD Retract
VAR_INPUT
END_VAR
END_METHOD

PROPERTY RetractAsserted : BOOL
END_PROPERTY

END_INTERFACE

// Interfaces/IExhaustable
INTERFACE IExhaustable EXTENDS ICylinder

METHOD Exhaust : BOOL
VAR_INPUT
END_VAR
END_METHOD

END_INTERFACE

// Interfaces/IExtendLowPressure
INTERFACE IExtendLowPressure EXTENDS ICylinder

METHOD ExtendLowPressure
VAR_INPUT
END_VAR
END_METHOD

PROPERTY ExtendLPAsserted : BOOL
END_PROPERTY

END_INTERFACE

// Interfaces/IInitializable
INTERFACE IInitializable EXTENDS IAllObjects

METHOD Initialize
VAR_INPUT
END_VAR
END_METHOD

END_INTERFACE

// Interfaces/IPositionableMotor
INTERFACE IPositionableMotor EXTENDS IAllObjects

PROPERTY CommandAcknowledged : BOOL        //Command acked from drive
END_PROPERTY

PROPERTY CurrentPosition : REAL        //Current motor position in Inches
END_PROPERTY

METHOD HomeNow
VAR_INPUT
END_VAR
END_METHOD

PROPERTY HomeRequired : BOOL
END_PROPERTY

PROPERTY Homing : BOOL
END_PROPERTY

PROPERTY InPosition : BOOL        //Motor is in position
END_PROPERTY

METHOD MoveDistance
VAR_INPUT
    distance : REAL;        //Distance to move in inches
    acceleration : INT;        //Acceleration in RPM/sec
    deceleration : INT;        //Deceleration in RPM/sec
    velocity : INT;            //Velocity in .25RPM
END_VAR
END_METHOD

METHOD MoveToPosition
VAR_INPUT
    position : REAL;        //Position to move to in inches
    acceleration : INT;        //Acceleration in RPM/sec
    deceleration : INT;        //Deceleration in RPM/sec
    velocity : INT;            //Velocity in .25RPM
END_VAR
END_METHOD

PROPERTY Moving : BOOL        //Motor is Moving
END_PROPERTY

METHOD Stop
VAR_INPUT
END_VAR
END_METHOD

END_INTERFACE

// Interfaces/IThreePositonCylinder
INTERFACE IThreePositonCylinder EXTENDS ICylinder

METHOD Exhaust
VAR_INPUT
END_VAR
END_METHOD

METHOD ExtendLowPressure
VAR_INPUT
END_VAR
END_METHOD

END_INTERFACE

// GetLibVersion
// This function has been automatically generated from the project information.
FUNCTION GetLibVersion : VERSION
VAR_INPUT
	
END_VAR

GetLibVersion.uiMajor := 0;
GetLibVersion.uiMinor := 9;
GetLibVersion.uiServicePack := 20;
GetLibVersion.uiPatch := 33;

END_FUNCTION

// GetLibVersionNumber
// This function has been automatically generated from the project information.
FUNCTION GetLibVersionNumber : DWORD
VAR_INPUT
	
END_VAR

GetLibVersionNumber := 594977;

END_FUNCTION

// ObjectHandling/FB_CollectionHandleMachineComponents
FUNCTION_BLOCK FB_CollectionHandleMachineComponents
VAR_INPUT
END_VAR
VAR
	Collection: ARRAY[0..GlobalObjects.MAX_COMPONENTS] OF IComponent; // object array
	ObjNames   : ARRAY[0..GlobalObjects.MAX_COMPONENTS] OF STRING;
	ActiveState : ARRAY[0..GlobalObjects.MAX_COMPONENTS] OF STRING;
	Ready : ARRAY[0..GlobalObjects.MAX_COMPONENTS] OF BOOL;
	InUse : ARRAY[0..GlobalObjects.MAX_COMPONENTS] OF BOOL;
	_ArrayOver   : BOOL;
	_BadObj      : INT;
	_DupeObj   : INT;
	_OverObj   : INT;
	_TotalObj   : UINT;

END_VAR

//	Function Block: FB_CollectionHandlerExecutable
//	Description: This collection handler stores executable FB's to an array 
//				 and has a method to execute them all on demand
//	Created by: Ben Hess
//	Created Date: Friday, September 7, 2018

METHOD AddObject
VAR_INPUT
	Obj : IComponent;
END_VAR
VAR
	I : UINT;
	J : UINT;
END_VAR
// Add the active fault to the array 
FOR J:= 0 TO _TotalObj DO
	IF Collection[J] = Obj THEN
		// object pointer matches - it's already in here
		RETURN;
	END_IF
END_FOR
   
IF _TotalObj < GlobalObjects.MAX_COMPONENTS THEN
	Collection[_TotalObj]:= Obj;
	ObjNames[_TotalObj]:= Obj.InstanceName;
	_TotalObj:= _TotalObj + 1;
ELSE
	_ArrayOver:= TRUE;
	_OverObj:= _OverObj + 1;
END_IF
END_METHOD

METHOD CheckIfAllHomed : BOOL
VAR_INPUT
END_VAR
VAR
	J : UINT;
	notHomed : BOOL;
END_VAR
// Go through list of homable components and return true if all are homed OR if component isn't active
FOR J:= 0 TO _TotalObj - 1 DO
	IF NOT CheckIfHomed(Collection[J]) THEN
		notHomed := TRUE;
	END_IF
END_FOR
CheckIfAllHomed := NOT notHomed;
END_METHOD

METHOD CheckIfAllReady : BOOL
VAR_INPUT
END_VAR
VAR
	J : UINT;
	notReady : BOOL;
END_VAR
// Go through list of homable components and return true if all are homed OR if component isn't active
FOR J:= 0 TO _TotalObj - 1 DO
	IF NOT CheckIfReady(Collection[J]) THEN
		notReady := TRUE;
	END_IF
END_FOR
CheckIfAllReady := NOT notReady;
END_METHOD

METHOD ForceHomeAll
VAR_INPUT
END_VAR
VAR
	Cast : IHomable;
	J : UINT;
END_VAR
// For each homable objest in the array, run its "HomeNow()" method
FOR J:= 0 TO _TotalObj - 1 DO
	IF (__QUERYINTERFACE(Collection[J], Cast)) THEN
		Cast.HomeNow();
	END_IF
END_FOR
END_METHOD

METHOD HomeAll
VAR_INPUT
END_VAR
VAR
	Cast : IHomable;
	J : UINT;
END_VAR
// For each homable objest in the array, run its "HomeNow()" method if object is not homed
FOR J:= 0 TO _TotalObj - 1 DO
	IF (__QUERYINTERFACE(Collection[J], Cast)) THEN
		IF NOT Cast.IsHomed THEN
			Cast.HomeNow();
		END_IF
	END_IF
END_FOR
END_METHOD

METHOD MakeReadyAll : BOOL
VAR
	J : UINT;
END_VAR
// Reset all components
FOR J:= 0 TO _TotalObj - 1 DO
	IF NOT Collection[J].Ready AND Collection[j].OptionActive THEN
		Collection[J].MakeReady();
	END_IF
END_FOR
END_METHOD

METHOD ResetAll
VAR_INPUT
END_VAR
VAR
	J : UINT;
END_VAR
// Reset all components
FOR J:= 0 TO _TotalObj - 1 DO
	Collection[J].Reset();
END_FOR
END_METHOD

METHOD UpdateInfo : BOOL
VAR_INPUT
END_VAR
VAR
	J : UINT;
END_VAR
FOR J:= 0 TO _TotalObj - 1 DO
		ActiveState[J]:= Collection[J].StateString;
		Ready[J] :=  Collection[J].Ready;
		InUse[J] := Collection[J].OptionActive AND Collection[J].OptionEnabled;
END_FOR
END_METHOD

END_FUNCTION_BLOCK

// ObjectHandling/FB_CollectionHandlerExecutable
FUNCTION_BLOCK FB_CollectionHandlerExecutable
VAR_INPUT
END_VAR
VAR
	Collection: ARRAY[0..GlobalObjects.MAX_EXECUTEABLE] OF IExecuteAutomatically; // object array
	ObjNames   : ARRAY[0..GlobalObjects.MAX_EXECUTEABLE] OF STRING;
	_ArrayOver   : BOOL;
	_BadObj      : INT;
	_DupeObj   : INT;
	_OverObj   : INT;
	_TotalObj   : UINT;
END_VAR

//	Function Block: FB_CollectionHandlerExecutable
//	Description: This collection handler stores executable FB's to an array 
//				 and has a method to execute them all on demand
//	Created by: Ben Hess
//	Created Date: Friday, September 7, 2018

METHOD AddObject
VAR_INPUT
	Obj   : IExecuteAutomatically;
END_VAR
VAR
	I   : UINT;
	J : UINT;
END_VAR
// Add the active fault to the array 
FOR J:= 0 TO _TotalObj DO
	IF Collection[J] = Obj THEN
		// object pointer matches - it's already in here
		RETURN;
	END_IF
END_FOR
   
IF _TotalObj < GlobalObjects.MAX_EXECUTEABLE THEN
	Collection[_TotalObj]:= Obj;
	ObjNames[_TotalObj]:= Obj.InstanceName;
	_TotalObj:= _TotalObj + 1;
ELSE
	_ArrayOver:= TRUE;
	_OverObj:= _OverObj + 1;
END_IF
END_METHOD

METHOD ExecuteAll
VAR_INPUT
END_VAR
VAR
	Cast : IExecuteAutomatically;
	J : UINT;
END_VAR
// For each executable objest in the array, run its "Execute()" method
FOR J:= 0 TO _TotalObj - 1 DO
	Collection[J].Execute();
END_FOR
END_METHOD

END_FUNCTION_BLOCK

// ObjectHandling/FB_CollectionHandlerExecutable
FUNCTION_BLOCK FB_CollectionHandlerExecutable
VAR_INPUT
END_VAR
VAR
	Collection: ARRAY[0..GlobalObjects.MAX_EXECUTEABLE] OF IExecuteAutomatically; // object array
	ObjNames   : ARRAY[0..GlobalObjects.MAX_EXECUTEABLE] OF STRING;
	_ArrayOver   : BOOL;
	_BadObj      : INT;
	_DupeObj   : INT;
	_OverObj   : INT;
	_TotalObj   : UINT;
END_VAR

//	Function Block: FB_CollectionHandlerExecutable
//	Description: This collection handler stores executable FB's to an array 
//				 and has a method to execute them all on demand
//	Created by: Ben Hess
//	Created Date: Friday, September 7, 2018

METHOD AddObject
VAR_INPUT
	Obj   : IExecuteAutomatically;
END_VAR
VAR
	I   : UINT;
	J : UINT;
END_VAR
// Add the active fault to the array 
FOR J:= 0 TO _TotalObj DO
	IF Collection[J] = Obj THEN
		// object pointer matches - it's already in here
		RETURN;
	END_IF
END_FOR
   
IF _TotalObj < GlobalObjects.MAX_EXECUTEABLE THEN
	Collection[_TotalObj]:= Obj;
	ObjNames[_TotalObj]:= Obj.InstanceName;
	_TotalObj:= _TotalObj + 1;
ELSE
	_ArrayOver:= TRUE;
	_OverObj:= _OverObj + 1;
END_IF
END_METHOD

METHOD ExecuteAll
VAR_INPUT
END_VAR
VAR
	Cast : IExecuteAutomatically;
	J : UINT;
END_VAR
// For each executable objest in the array, run its "Execute()" method
FOR J:= 0 TO _TotalObj - 1 DO
	IF (__QUERYINTERFACE(Collection[J], Cast)) THEN
		Cast.Execute();
	ELSE 
		RETURN;
	END_IF
END_FOR
END_METHOD

END_FUNCTION_BLOCK

// Testing/HelperFunctions/CheckIfHomed
FUNCTION CheckIfHomed : BOOL
VAR_INPUT
	Component : IComponent;
END_VAR
VAR
	homableDevice : IHomable;
END_VAR

//	Function: CheckIfHomed()
//	Description: Helper function
//				 Pass in a component - if it has a homable motor, and is not yet homed, start homing
//	Created by: Ben Hess
//	Created Date: May 16th, 2019

IF (__QUERYINTERFACE(Component, homableDevice)) THEN
	IF homableDevice.IsHomed OR NOT Component.OptionActive THEN
		CheckIfHomed := TRUE;
	ELSE 
		RETURN;
	END_IF
ELSE
	CheckIfHomed := TRUE;
END_IF

END_FUNCTION

// Testing/Motors/IHomable
INTERFACE IHomable EXTENDS IAllObjects

END_INTERFACE

// Testing/HelperFunctions/CheckIfReady
FUNCTION CheckIfReady : BOOL
VAR_INPUT
	Component : IComponent;
END_VAR
VAR
END_VAR

//	Function: CheckIfReady()
//	Description: Helper function
//				 Pass in a component - if it has a homable motor, and is not yet homed, start homing
//	Created by: Ben Hess
//	Created Date: June 13th, 2020

IF Component.Ready OR NOT Component.OptionActive THEN
	CheckIfReady := TRUE;
ELSE
	RETURN;
END_IF

END_FUNCTION

// ObjectHandling/FB_CollectionHandlerActiveFaults
FUNCTION_BLOCK FB_CollectionHandlerActiveFaults
VAR_INPUT
END_VAR
VAR
	Collection: ARRAY[0..GlobalObjects.MAX_FAULTS] OF IFault; // object array
	ObjNames   : ARRAY[0..GlobalObjects.MAX_FAULTS] OF STRING;
	ObjIds	: ARRAY[0..GlobalObjects.MAX_FAULTS] OF DINT;
	_ArrayOver   : BOOL;
	_BadObj      : INT;
	_DupeObj   : INT;
	_OverObj   : INT;
	_TotalObj   : UINT;
END_VAR

VAR_OUTPUT
	faultActive : BOOL;
END_VAR

//	Function Block: FB_CollectionHandlerActiveFaults
//	Description: This collection handler adds and removes active faults to an array
//				 The add and remove methods are called from FB_Fault
//	Created by: Tom Jacobs
//	Created Date: Friday, September 7, 2018

METHOD AckAll
VAR_INPUT
END_VAR
VAR
	Cast : IFault;
	Fault : IFault;
	J : UINT;
END_VAR
// For each active fault in the array, ack it.
IF _TotalObj <=0 THEN
	RETURN;
END_IF
FOR J:= 0 TO _TotalObj - 1 DO
		Collection[J].Ack();
END_FOR
END_METHOD

METHOD AddObject
VAR_INPUT
	Obj   : IFault;
END_VAR
VAR
	I   : UINT;
	J : UINT;
END_VAR
// Add the active fault to the array 
FOR J:= 0 TO _TotalObj DO
	IF Collection[J] = Obj THEN
		// object pointer matches - it's already in here
		RETURN;
	END_IF
END_FOR
   
IF _TotalObj < GlobalObjects.MAX_FAULTS THEN
	Collection[_TotalObj]:= Obj;
	ObjNames[_TotalObj]:= Obj.InstanceName;
	ObjIDs[_TotalObj]:= Obj.FaultID;
	_TotalObj:= _TotalObj + 1;
ELSE
	_ArrayOver:= TRUE;
	_OverObj:= _OverObj + 1;
END_IF
GlobalObjects.CollectionOfFaults.FaultUpdateForHMI();
faultActive := TRUE;
END_METHOD

METHOD RemoveObject
VAR_INPUT
	Obj   : IFault;
END_VAR

VAR
	I   : UINT;
	J : UINT;
END_VAR
FOR I:= 0 TO _TotalObj DO
	IF Collection[I] = Obj THEN
		// object pointer matches - get rid of it
		FOR J := I TO _TotalObj DO
			Collection[J] := Collection[J+1];
			ObjNames[J]:= ObjNames[J+1];
			ObjIDs[J]:= ObjIDs[J+1];
		END_FOR
		_TotalObj := _TotalObj - 1;

		IF _TotalObj = 0 THEN
			GlobalObjects.CollectionOfFaults.FaultUpdateForHMI();
			faultActive := FALSE;
		END_IF
		RETURN;
	END_IF
END_FOR
END_METHOD

END_FUNCTION_BLOCK

// ObjectHandling/FB_CollectionHandlerActiveFaults
FUNCTION_BLOCK FB_CollectionHandlerActiveFaults
VAR_INPUT
END_VAR
VAR
	Collection: ARRAY[0..GlobalObjects.MAX_FAULTS] OF IFault; // object array
	ObjNames   : ARRAY[0..GlobalObjects.MAX_FAULTS] OF STRING;
	_ArrayOver   : BOOL;
	_BadObj      : INT;
	_DupeObj   : INT;
	_OverObj   : INT;
END_VAR
VAR_OUTPUT
	totalObj   : UINT;
	faultActive : BOOL;
END_VAR

//	Function Block: FB_CollectionHandlerActiveFaults
//	Description: This collection handler adds and removes active faults to an array
//				 The add and remove methods are called from FB_Fault
//	Created by: Tom Jacobs
//	Created Date: Friday, September 7, 2018

METHOD AckAll
VAR_INPUT
END_VAR
VAR
	Cast : IFault;
	Fault : IFault;
	J : UINT;
END_VAR
// For each active fault in the array, ack it.
FOR J:= 0 TO totalObj - 1 DO
	IF (__QUERYINTERFACE(Collection[J], Cast)) THEN
		Cast.Ack();
	ELSE 
		RETURN;
	END_IF
END_FOR
END_METHOD

METHOD AddObject
VAR_INPUT
	Obj   : IFault;
END_VAR
VAR
	I   : UINT;
	J : UINT;
END_VAR
// Add the active fault to the array 
FOR J:= 0 TO totalObj DO
	IF Collection[J] = Obj THEN
		// object pointer matches - it's already in here
		RETURN;
	END_IF
END_FOR
   
IF totalObj < GlobalObjects.MAX_FAULTS THEN
	Collection[totalObj]:= Obj;
	ObjNames[totalObj]:= Obj.InstanceName;
	totalObj:= totalObj + 1;
ELSE
	_ArrayOver:= TRUE;
	_OverObj:= _OverObj + 1;
END_IF
faultActive := TRUE;
END_METHOD

METHOD RemoveObject
VAR_INPUT
	Obj   : IFault;
END_VAR

VAR
	I   : UINT;
	J : UINT;
END_VAR
FOR I:= 0 TO totalObj DO
	IF Collection[I] = Obj THEN
		// object pointer matches - get rid of it
		FOR J := I TO totalObj DO
			Collection[J] := Collection[J+1];
			ObjNames[J]:= ObjNames[J+1]; 
		END_FOR
		totalObj := totalObj - 1;
		IF totalObj = 0 THEN
			faultActive := FALSE;
		END_IF
		RETURN;
	END_IF
END_FOR
END_METHOD

END_FUNCTION_BLOCK

// FBs/Fault/FB_Fault
FUNCTION_BLOCK FINAL FB_Fault IMPLEMENTS IFault, ILoggable, IExecuteAutomatically
VAR_INPUT
	ackCommand : BOOL;
	faultTrigger : BOOL;
END_VAR
VAR_OUTPUT
	acknowledged : BOOL;
	active : BOOL;
END_VAR
VAR
	_acked : BOOL;
	_active : BOOL;
	_logger : IMachineLogger;
	_faultTriggerONS : FB_ONS;
	_ackCommandONS : FB_ONS;
	_activeONS : FB_ONS;
	_instanceName : STRING;
END_VAR
VAR_IN_OUT
END_VAR

END_FUNCTION_BLOCK

// ObjectHandling/FB_CollectionHandlerAll
FUNCTION_BLOCK FINAL FB_CollectionHandlerAll
VAR_INPUT
END_VAR
VAR
	Collection: ARRAY[0..GlobalObjects.MAX_OBJECTS] OF IAllObjects; // object array
	ObjNames   : ARRAY[0..GlobalObjects.MAX_OBJECTS] OF STRING;
	_ArrayOver   : BOOL;
	_BadObj      : INT;
	_DupeObj   : INT;
	_OverObj   : INT;
	_TotalObj   : UINT;
END_VAR

METHOD FINAL AddObject
VAR_INPUT
	Obj   : IAllObjects;
END_VAR
VAR
	AnyObject : IAllObjects;
	Fault : IFault;
	Cylinder : ICylinder;
	PositionableMotor : IPositionableMotor;
	Logger : IMachineLogger;
	Loggable : ILoggable;
	Executable : IExecuteAutomatically;
	Initializable : IInitializable;
	J   : UINT;
END_VAR
IF (__QUERYINTERFACE(Obj, AnyObject)) THEN
   // make sure haven't already added this object
   FOR J:= 1 TO _TotalObj DO
      IF Collection[J] = AnyObject THEN
         // object pointer matches - dupe!
         _DupeObj:= _DupeObj + 1;
         RETURN;
      END_IF
   END_FOR
   
   IF _TotalObj < GlobalObjects.MAX_OBJECTS THEN
      Collection[_TotalObj]:= AnyObject;
      ObjNames[_TotalObj]:= Obj.InstanceName;
	   _TotalObj:= _TotalObj + 1;
   ELSE
      _ArrayOver:= TRUE;
      _OverObj:= _OverObj + 1;
   END_IF
ELSE
   _BadObj:= _BadObj + 1;
END_IF

// Add object to proper collection based on its interfaces
IF (__QUERYINTERFACE(Obj, Fault)) THEN
	GlobalObjects.CollectionOfFaults.AddObject(Fault);
END_IF

// IF (__QUERYINTERFACE(Obj, Cylinder)) THEN
// 	GlobalObjects.CollectionOfCylinders.AddObject(Cylinder);
// END_IF
// 
// IF (__QUERYINTERFACE(Obj, PositionableMotor)) THEN
// 	GlobalObjects.CollectionOfPositionableMotors.AddObject(PositionableMotor);
// END_IF

IF (__QUERYINTERFACE(Obj, Logger)) THEN
	GlobalObjects.CollectionOfLogs.AddObject(Logger);
END_IF

IF (__QUERYINTERFACE(Obj, Loggable)) THEN
	GlobalObjects.CollectionOfLoggable.AddObject(Loggable);
END_IF

IF (__QUERYINTERFACE(Obj, Executable)) THEN
	GlobalObjects.CollectionOfExecutable.AddObject(Executable);
END_IF

IF (__QUERYINTERFACE(Obj, Initializable)) THEN
	GlobalObjects.CollectionOfInitialzable.AddObject(Initializable);
END_IF
END_METHOD

END_FUNCTION_BLOCK

// ObjectHandling/FB_CollectionHandlerCylinders
FUNCTION_BLOCK FB_CollectionHandlerCylinders
VAR_INPUT
END_VAR
VAR
	Collection: ARRAY[0..GlobalObjects.MAX_CYLINDERS] OF ICylinder; // object array
	ObjNames   : ARRAY[0..GlobalObjects.MAX_CYLINDERS] OF STRING;
	_ArrayOver   : BOOL;
	_BadObj      : INT;
	_DupeObj   : INT;
	_OverObj   : INT;
	_TotalObj   : UINT;
END_VAR

METHOD AddObject
VAR_INPUT
	Obj   : ICylinder;
END_VAR
VAR
	Cast: ICylinder;
	J   : UINT;
END_VAR
FOR J:= 0 TO _TotalObj DO
	IF Collection[J] = Obj THEN
		// object pointer matches - dupe!
		_DupeObj:= _DupeObj + 1;
		RETURN;
	END_IF
END_FOR
   
IF _TotalObj < GlobalObjects.MAX_CYLINDERS THEN
	Collection[_TotalObj]:= Obj;
	ObjNames[_TotalObj]:= Obj.InstanceName;
	_TotalObj:= _TotalObj + 1;
ELSE
	_ArrayOver:= TRUE;
	_OverObj:= _OverObj + 1;
END_IF
END_METHOD

END_FUNCTION_BLOCK

// ObjectHandling/FB_CollectionHandlerFaults
FUNCTION_BLOCK FB_CollectionHandlerFaults
VAR_INPUT
END_VAR
VAR
	Collection: ARRAY[0..GlobalObjects.MAX_FAULTS] OF IFault; // object array
	ObjNames   : ARRAY[0..GlobalObjects.MAX_FAULTS] OF STRING;
	faults : ARRAY[0..GlobalObjects.MAX_FAULTS] OF HMIFaultType;
	_ArrayOver   : BOOL;
	_BadObj      : INT;
	_DupeObj   : INT;
	_OverObj   : INT;
	_TotalObj   : UINT;
	_InitFaultList : BOOL;
END_VAR

METHOD AckAll
VAR_INPUT
END_VAR
VAR
	Cast : IFault;
	Fault : IFault;
	J : UINT;
END_VAR
// For each active fault in the array, ack it.
IF _TotalObj <=0 THEN
	RETURN;
END_IF
FOR J:= 0 TO _TotalObj - 1 DO
		Collection[J].Ack();
END_FOR
END_METHOD

METHOD AddObject
VAR_INPUT
	Obj   : IFault;
END_VAR
VAR
	J   : UINT;
END_VAR
FOR J:= 0 TO _TotalObj DO
	IF Collection[J] = Obj THEN
		// object pointer matches - dupe!
		_DupeObj:= _DupeObj + 1;
		RETURN;
	END_IF
END_FOR
   
IF _TotalObj < GlobalObjects.MAX_FAULTS THEN
	Collection[_TotalObj]:= Obj;
	ObjNames[_TotalObj]:= Obj.InstanceName;
	_TotalObj:= _TotalObj + 1;
ELSE
	_ArrayOver:= TRUE;
	_OverObj:= _OverObj + 1;
END_IF
END_METHOD

METHOD FaultUpdateForHMI
VAR_INPUT
END_VAR
VAR
	I : UINT;
END_VAR
FOR I:= 0 TO _TotalObj - 1 DO
	IF NOT _InitFaultList THEN
		faults[I].name := Collection[I].InstanceName;
	END_IF
	faults[I].active := Collection[I].FaultActive;
END_FOR
_InitFaultList := TRUE;
END_METHOD

END_FUNCTION_BLOCK

// ObjectHandling/FB_CollectionHandlerFaults
FUNCTION_BLOCK FB_CollectionHandlerFaults
VAR_INPUT
END_VAR
VAR
	Collection: ARRAY[0..GlobalObjects.MAX_FAULTS] OF IFault; // object array
	ObjNames   : ARRAY[0..GlobalObjects.MAX_FAULTS] OF STRING;
	_ArrayOver   : BOOL;
	_BadObj      : INT;
	_DupeObj   : INT;
	_OverObj   : INT;
	_TotalObj   : UINT;
END_VAR

METHOD AckAll
VAR_INPUT
END_VAR
VAR
	J : UINT;
END_VAR
FOR J:= 0 TO _TotalObj - 1 DO
	Collection[J].Ack();
END_FOR
END_METHOD

METHOD AddObject
VAR_INPUT
	Obj   : IFault;
END_VAR
VAR
	J   : UINT;
END_VAR
FOR J:= 0 TO _TotalObj DO
	IF Collection[J] = Obj THEN
		// object pointer matches - dupe!
		_DupeObj:= _DupeObj + 1;
		RETURN;
	END_IF
END_FOR
   
IF _TotalObj < GlobalObjects.MAX_FAULTS THEN
	Collection[_TotalObj]:= Obj;
	ObjNames[_TotalObj]:= Obj.InstanceName;
	_TotalObj:= _TotalObj + 1;
ELSE
	_ArrayOver:= TRUE;
	_OverObj:= _OverObj + 1;
END_IF
END_METHOD

END_FUNCTION_BLOCK

// ObjectHandling/FB_CollectionHandlerInitializable
FUNCTION_BLOCK FB_CollectionHandlerInitializable
VAR_INPUT

END_VAR
VAR
	Collection: ARRAY[0..GlobalObjects.MAX_LOGGABLE] OF IInitializable; // object array
	ObjNames   : ARRAY[0..GlobalObjects.MAX_LOGGABLE] OF STRING;
	_ArrayOver   : BOOL;
	_BadObj      : INT;
	_DupeObj   : INT;
	_OverObj   : INT;
	_TotalObj   : UINT;
END_VAR

//	Function Block: FB_CollectionHandlerLoggable
//	Description: This collection handler takes in loggable objects and registers them with a logger.  The FirstScan function should trigger the 
//				 RegisterAll() method to register all loggable objects with a logger
//	Created by: Ben Hess
//	Created Date: Tuesday, September 11, 2018

METHOD AddObject
VAR_INPUT
	Obj   : IInitializable;
END_VAR
VAR
	J   : UINT;
END_VAR
FOR J:= 0 TO _TotalObj DO
	IF Collection[J] = Obj THEN
		// object pointer matches - dupe!
		_DupeObj:= _DupeObj + 1;
		RETURN;
	END_IF
END_FOR
   
IF _TotalObj < GlobalObjects.MAX_LOGGABLE THEN
	Collection[_TotalObj]:= Obj;
	ObjNames[_TotalObj]:= Obj.InstanceName;
	_TotalObj:= _TotalObj + 1;
ELSE
	_ArrayOver:= TRUE;
	_OverObj:= _OverObj + 1;
END_IF
END_METHOD

METHOD InitializeAll
VAR_INPUT
	
END_VAR
VAR
	J : UINT;
	Cast : IInitializable;
END_VAR
FOR J:= 0 TO _TotalObj - 1 DO
	IF (__QUERYINTERFACE(Collection[J], Cast)) THEN
		Cast.Initialize();
	ELSE 
		RETURN;
	END_IF
END_FOR
END_METHOD

END_FUNCTION_BLOCK

// ObjectHandling/FB_CollectionHandlerLoggable
FUNCTION_BLOCK FB_CollectionHandlerLoggable
VAR_INPUT

END_VAR
VAR
	Collection: ARRAY[0..GlobalObjects.MAX_LOGGABLE] OF ILoggable; // object array
	ObjNames   : ARRAY[0..GlobalObjects.MAX_LOGGABLE] OF STRING;
	_ArrayOver   : BOOL;
	_BadObj      : INT;
	_DupeObj   : INT;
	_OverObj   : INT;
	_TotalObj   : UINT;
	_internalLogger : REFERENCE TO IMachineLogger;
END_VAR

//	Function Block: FB_CollectionHandlerLoggable
//	Description: This collection handler takes in loggable objects and registers them with a logger.  The FirstScan function should trigger the 
//				 RegisterAll() method to register all loggable objects with a logger
//	Created by: Ben Hess
//	Created Date: Tuesday, September 11, 2018

METHOD AddObject
VAR_INPUT
	Obj   : ILoggable;
END_VAR
VAR
	J   : UINT;
END_VAR
FOR J:= 0 TO _TotalObj DO
	IF Collection[J] = Obj THEN
		// object pointer matches - dupe!
		_DupeObj:= _DupeObj + 1;
		RETURN;
	END_IF
END_FOR
   
IF _TotalObj < GlobalObjects.MAX_LOGGABLE THEN
	Collection[_TotalObj]:= Obj;
	ObjNames[_TotalObj]:= Obj.InstanceName;
	_TotalObj:= _TotalObj + 1;
ELSE
	_ArrayOver:= TRUE;
	_OverObj:= _OverObj + 1;
END_IF
END_METHOD

METHOD RegisterAll
VAR_INPUT
	internalLogger : IMachineLogger;
END_VAR
VAR
	I   : UINT;
	J : UINT;
	cast : ILoggable;
END_VAR
FOR J:= 0 TO _TotalObj - 1 DO
	IF (__QUERYINTERFACE(Collection[J], Cast)) THEN
		cast.RegisterLogger(internalLogger := internalLogger);
	ELSE
		RETURN;
	END_IF
END_FOR
END_METHOD

END_FUNCTION_BLOCK

// ObjectHandling/FB_CollectionHandlerLoggable
FUNCTION_BLOCK FB_CollectionHandlerLoggable
VAR_INPUT

END_VAR
VAR
	Collection: ARRAY[0..GlobalObjects.MAX_LOGGABLE] OF ILoggable; // object array
	ObjNames   : ARRAY[0..GlobalObjects.MAX_LOGGABLE] OF STRING;
	_ArrayOver   : BOOL;
	_BadObj      : INT;
	_DupeObj   : INT;
	_OverObj   : INT;
	_TotalObj   : UINT;
	_internalLogger : REFERENCE TO IMachineLogger;
END_VAR

//	Function Block: FB_CollectionHandlerLoggable
//	Description: This collection handler takes in loggable objects and registers them with a logger.  The FirstScan function should trigger the 
//				 RegisterAll() method to register all loggable objects with a logger
//	Created by: Ben Hess
//	Created Date: Tuesday, September 11, 2018

METHOD AddObject
VAR_INPUT
	Obj   : ILoggable;
END_VAR
VAR
	J   : UINT;
END_VAR
FOR J:= 0 TO _TotalObj DO
	IF Collection[J] = Obj THEN
		// object pointer matches - dupe!
		_DupeObj:= _DupeObj + 1;
		RETURN;
	END_IF
END_FOR
   
IF _TotalObj < GlobalObjects.MAX_LOGGABLE THEN
	Collection[_TotalObj]:= Obj;
	ObjNames[_TotalObj]:= Obj.InstanceName;
	_TotalObj:= _TotalObj + 1;
ELSE
	_ArrayOver:= TRUE;
	_OverObj:= _OverObj + 1;
END_IF
END_METHOD

METHOD RegisterAll
VAR_INPUT
	internalLogger : IMachineLogger;
END_VAR
VAR
	I   : UINT;
	J : UINT;
	cast : ILoggable;
END_VAR
FOR J:= 0 TO _TotalObj - 1 DO
	IF (__QUERYINTERFACE(Collection[J], Cast)) THEN
		cast.RegisterLogger(internalLogger := internalLogger);
	ELSE
		RETURN;
	END_IF
END_FOR
END_METHOD

END_FUNCTION_BLOCK

// ObjectHandling/FB_CollectionHandlerInitializable
FUNCTION_BLOCK FB_CollectionHandlerInitializable
VAR_INPUT

END_VAR
VAR
	Collection: ARRAY[0..GlobalObjects.MAX_LOGGABLE] OF IInitializable; // object array
	ObjNames   : ARRAY[0..GlobalObjects.MAX_LOGGABLE] OF STRING;
	_ArrayOver   : BOOL;
	_BadObj      : INT;
	_DupeObj   : INT;
	_OverObj   : INT;
	_TotalObj   : UINT;
END_VAR

//	Function Block: FB_CollectionHandlerLoggable
//	Description: This collection handler takes in loggable objects and registers them with a logger.  The FirstScan function should trigger the 
//				 RegisterAll() method to register all loggable objects with a logger
//	Created by: Ben Hess
//	Created Date: Tuesday, September 11, 2018

METHOD AddObject
VAR_INPUT
	Obj   : IInitializable;
END_VAR
VAR
	J   : UINT;
END_VAR
FOR J:= 0 TO _TotalObj DO
	IF Collection[J] = Obj THEN
		// object pointer matches - dupe!
		_DupeObj:= _DupeObj + 1;
		RETURN;
	END_IF
END_FOR
   
IF _TotalObj < GlobalObjects.MAX_LOGGABLE THEN
	Collection[_TotalObj]:= Obj;
	ObjNames[_TotalObj]:= Obj.InstanceName;
	_TotalObj:= _TotalObj + 1;
ELSE
	_ArrayOver:= TRUE;
	_OverObj:= _OverObj + 1;
END_IF
END_METHOD

METHOD InitializeAll
VAR_INPUT
	
END_VAR
VAR
	J : UINT;
	Cast : IInitializable;
END_VAR
FOR J:= 0 TO _TotalObj - 1 DO
	IF (__QUERYINTERFACE(Collection[J], Cast)) THEN
		Cast.Initialize();
	ELSE 
		RETURN;
	END_IF
END_FOR
END_METHOD

END_FUNCTION_BLOCK

// ObjectHandling/FB_CollectionHandlerLogs
FUNCTION_BLOCK FB_CollectionHandlerLogs
VAR_INPUT
END_VAR
VAR
	Collection: ARRAY[0..GlobalObjects.MAX_LOGS] OF IMachineLogger; // object array
	ObjNames   : ARRAY[0..GlobalObjects.MAX_LOGS] OF STRING;
	_ArrayOver   : BOOL;
	_BadObj      : INT;
	_DupeObj   : INT;
	_OverObj   : INT;
	_TotalObj   : UINT;
END_VAR

METHOD AddObject
VAR_INPUT
	Obj   : IMachineLogger;
END_VAR
VAR
	J   : UINT;
END_VAR
FOR J:= 0 TO _TotalObj DO
	IF Collection[J] = Obj THEN
		// object pointer matches - dupe!
		_DupeObj:= _DupeObj + 1;
		RETURN;
	END_IF
END_FOR
   
IF _TotalObj < GlobalObjects.MAX_LOGS THEN
	Collection[_TotalObj]:= Obj;
	ObjNames[_TotalObj]:= Obj.InstanceName;
	_TotalObj:= _TotalObj + 1;
ELSE
	_ArrayOver:= TRUE;
	_OverObj:= _OverObj + 1;
END_IF
END_METHOD

END_FUNCTION_BLOCK

// ObjectHandling/FB_CollectionHandlerLogs
FUNCTION_BLOCK FB_CollectionHandlerLogs
VAR_INPUT
END_VAR
VAR
	Collection: ARRAY[0..GlobalObjects.MAX_LOGS] OF IMachineLogger; // object array
	ObjNames   : ARRAY[0..GlobalObjects.MAX_LOGS] OF STRING;
	_ArrayOver   : BOOL;
	_BadObj      : INT;
	_DupeObj   : INT;
	_OverObj   : INT;
	_TotalObj   : UINT;
END_VAR

METHOD AddObject
VAR_INPUT
	Obj   : IMachineLogger;
END_VAR
VAR
	J   : UINT;
END_VAR
FOR J:= 0 TO _TotalObj DO
	IF Collection[J] = Obj THEN
		// object pointer matches - dupe!
		_DupeObj:= _DupeObj + 1;
		RETURN;
	END_IF
END_FOR
   
IF _TotalObj < GlobalObjects.MAX_LOGS THEN
	Collection[_TotalObj]:= Obj;
	ObjNames[_TotalObj]:= Obj.InstanceName;
	_TotalObj:= _TotalObj + 1;
ELSE
	_ArrayOver:= TRUE;
	_OverObj:= _OverObj + 1;
END_IF
END_METHOD

END_FUNCTION_BLOCK

// ObjectHandling/FB_CollectionHandlerPositionableMotors
FUNCTION_BLOCK FB_CollectionHandlerPositionableMotors
VAR_INPUT
END_VAR
VAR
	Collection: ARRAY[0..GlobalObjects.MAX_MOTORS] OF IPositionableMotor; // object array
	ObjNames   : ARRAY[0..GlobalObjects.MAX_MOTORS] OF STRING;
	_ArrayOver   : BOOL;
	_BadObj      : INT;
	_DupeObj   : INT;
	_OverObj   : INT;
	_TotalObj   : UINT;
END_VAR

METHOD AddObject
VAR_INPUT
	Obj   : IPositionableMotor;
END_VAR
VAR
	J   : UINT;
END_VAR
FOR J:= 0 TO _TotalObj DO
	IF Collection[J] = Obj THEN
		// object pointer matches - dupe!
		_DupeObj:= _DupeObj + 1;
		RETURN;
	END_IF
END_FOR
   
IF _TotalObj < GlobalObjects.MAX_MOTORS THEN
	Collection[_TotalObj]:= Obj;
	ObjNames[_TotalObj]:= Obj.InstanceName;
	_TotalObj:= _TotalObj + 1;
ELSE
	_ArrayOver:= TRUE;
	_OverObj:= _OverObj + 1;
END_IF
END_METHOD

END_FUNCTION_BLOCK

// ObjectHandling/IResettable
INTERFACE IResettable EXTENDS IAllObjects

END_INTERFACE

// GetCompany
// This function has been automatically generated from the project information.
{attribute 'signature_flag' := '1073741824'}
{attribute 'register_in_runtime'}
FUNCTION GetCompany : WSTRING
VAR_INPUT
	
END_VAR

GetCompany := "Sharp Packaging";

END_FUNCTION

// GetTextProperty2
// This function has been automatically generated from the project information.
{attribute 'signature_flag' := '1073741824'}
{attribute 'register_in_runtime'}
FUNCTION GetTextProperty2 : POINTER TO WSTRING
VAR_INPUT
	stKey: WSTRING;
END_VAR

IF stKey = "Author" THEN
	GetTextProperty2 := ADR("Ben Hess");
ELSIF stKey = "Company" THEN
	GetTextProperty2 := ADR("Sharp Packaging");
ELSIF stKey = "CompiledLibraryCompatibilityVersion" THEN
	GetTextProperty2 := ADR("CODESYS V3.5 SP16");
ELSIF stKey = "Project" THEN
	GetTextProperty2 := ADR("AlphaController");
ELSIF stKey = "Title" THEN
	GetTextProperty2 := ADR("");
ELSIF stKey = "VersionPostfix" THEN
	GetTextProperty2 := ADR("-alpha/master");
ELSE
	GetTextProperty2 := ADR("");
END_IF

END_FUNCTION

// GetTextProperty
// This function has been automatically generated from the project information.
{attribute 'signature_flag' := '1073741824'}
{attribute 'register_in_runtime'}
FUNCTION GetTextProperty : WSTRING
VAR_INPUT
	stKey: WSTRING;
END_VAR

IF stKey = "Author" THEN
	GetTextProperty := "Ben Hess";
ELSIF stKey = "Company" THEN
	GetTextProperty := "Sharp Packaging";
ELSIF stKey = "CompiledLibraryCompatibilityVersion" THEN
	GetTextProperty := "CODESYS V3.5 SP16";
ELSIF stKey = "Project" THEN
	GetTextProperty := "AlphaController";
ELSIF stKey = "Title" THEN
	GetTextProperty := "";
ELSIF stKey = "VersionPostfix" THEN
	GetTextProperty := "-alpha/master";
ELSE
	GetTextProperty := "";
END_IF

END_FUNCTION

// GetTitle
// This function has been automatically generated from the project information.
{attribute 'signature_flag' := '1073741824'}
{attribute 'register_in_runtime'}
FUNCTION GetTitle : WSTRING
VAR_INPUT
	
END_VAR

GetTitle := "";

END_FUNCTION

// GetVersion
// This function has been automatically generated from the project information.
{attribute 'signature_flag' := '1073741824'}
{attribute 'register_in_runtime'}
FUNCTION GetVersion : VERSION
VAR_INPUT
	
END_VAR

GetVersion.uiMajor := 0;
GetVersion.uiMinor := 9;
GetVersion.uiServicePack := 20;
GetVersion.uiPatch := 33;

END_FUNCTION

// GetVersionProperty
// This function has been automatically generated from the project information.
{attribute 'signature_flag' := '1073741824'}
{attribute 'register_in_runtime'}
FUNCTION GetVersionProperty : VERSION
VAR_INPUT
	stKey: WSTRING;
END_VAR

IF stKey = "Version" THEN
	GetVersionProperty.uiMajor := 0;
	GetVersionProperty.uiMinor := 9;
	GetVersionProperty.uiServicePack := 20;
	GetVersionProperty.uiPatch := 33;
ELSE
	GetVersionProperty.uiMajor := 0;
	GetVersionProperty.uiMinor := 0;
	GetVersionProperty.uiServicePack := 0;
	GetVersionProperty.uiPatch := 0;
END_IF

END_FUNCTION

// Testing/FB_MultiUnitTest
(*
{attribute 'test' := 'multitest'}
{attribute 'testcasename':='Monostable Multivibrator'}
{attribute 'testcategory':='Basics'}
{attribute 'testcasetimeout':='360000'}
*)
FUNCTION_BLOCK FB_MultiUnitTest EXTENDS CBM.EtrigA
VAR_INPUT
	xGetTestInfo : BOOL;
    diTestCaseIndex : DINT;
END_VAR
VAR_OUTPUT
    sTestCaseName : STRING;
	sTestCaseCategories : STRING;
    diTestCaseCount : DINT;
    diTestCaseTimeout : DINT;
    sInfo : STRING;
	eError : UnitTestErrors;
    sError : STRING;
    eFailureMode : TM.FAILUREMODE;
END_VAR
VAR
	
END_VAR

{attribute 'hide'}
METHOD prvAbort : BOOL

SUPER^.prvAbort();

xAbortInProgress := FALSE;
END_METHOD

{attribute 'hide'}
METHOD prvCyclicAction : BOOL
SUPER^.prvCyclicAction();

CASE diTestCaseIndex OF
    0: 	IF THIS^.xGetTestInfo THEN
            THIS^.sTestCaseName := 'Step 1: ';
            THIS^.sTestCaseCategories := 'General';
            THIS^.diTestCaseTimeout := 3000;
			xDone := TRUE;
		ELSE
			(*TEST SOMETHING HERE*)
			IF (*CONNDITION*) FALSE THEN
				 xDone := TRUE;
			ELSE
				THIS^.sError := '';
				xError := TRUE;
				eError := UnitTestErrors.Failure;
            	eFailureMode := TM.FAILUREMODE.AbortTestCase;
                iError := 1;
			END_IF
        END_IF
    1: 	IF THIS^.xGetTestInfo THEN
            THIS^.sTestCaseName := 'Step 2: ';
            THIS^.sTestCaseCategories := 'General';
            THIS^.diTestCaseTimeout := 3000;
			xDone := TRUE;
		ELSE
			(*TEST SOMETHING HERE*)
			IF (*CONNDITION*) FALSE THEN
				 xDone := TRUE;
			ELSE
				THIS^.sError := '';
				xError := TRUE;
				eError := UnitTestErrors.Failure;
            	eFailureMode := TM.FAILUREMODE.AbortTestCase;
                iError := 1;
			END_IF
        END_IF
	   
	2: 	IF THIS^.xGetTestInfo THEN
            THIS^.sTestCaseName := 'Step 3: ';
            THIS^.sTestCaseCategories := 'General';
            THIS^.diTestCaseTimeout := 3000;
			xDone := TRUE;
		ELSE
			(*TEST SOMETHING HERE*)
			IF (*CONNDITION*) THEN
				 xDone := TRUE;
			ELSE
				THIS^.sError := '';
				xError := TRUE;
				eError := UnitTestErrors.Failure;
            	eFailureMode := TM.FAILUREMODE.AbortTestCase;
                iError := 1;
			END_IF
        END_IF

   	3: 	IF THIS^.xGetTestInfo THEN
            THIS^.sTestCaseName := 'Step 4: ';
            THIS^.sTestCaseCategories := 'General';
            THIS^.diTestCaseTimeout := 3000;
			xDone := TRUE;
		ELSE
			(*TEST SOMETHING HERE*)
			IF (*CONNDITION*) FALSE THEN
				 xDone := TRUE;
			ELSE
				THIS^.sError := '';
				xError := TRUE;
				eError := UnitTestErrors.Failure;
            	eFailureMode := TM.FAILUREMODE.AbortTestCase;
                iError := 1;
			END_IF
        END_IF
	   
	4: 	IF THIS^.xGetTestInfo THEN
            THIS^.sTestCaseName := 'Step 5: ';
            THIS^.sTestCaseCategories := 'General';
            THIS^.diTestCaseTimeout := 3000;
			xDone := TRUE;
		ELSE
			(*TEST SOMETHING HERE*)
			IF (*CONNDITION*) FALSE THEN
				 xDone := TRUE;
			ELSE
				THIS^.sError := '';
				xError := TRUE;
				eError := UnitTestErrors.Failure;
            	eFailureMode := TM.FAILUREMODE.AbortTestCase;
                iError := 1;
			END_IF
        END_IF
		
	5: 	IF THIS^.xGetTestInfo THEN
            THIS^.sTestCaseName := 'Step 6: ';
            THIS^.sTestCaseCategories := 'General';
            THIS^.diTestCaseTimeout := 3000;
			xDone := TRUE;
		ELSE
			(*TEST SOMETHING HERE*)
			IF (*CONNDITION*) FALSE THEN
				 xDone := TRUE;
			ELSE
				THIS^.sError := '';
				xError := TRUE;
				eError := UnitTestErrors.Failure;
            	eFailureMode := TM.FAILUREMODE.AbortTestCase;
                iError := 1;
			END_IF
        END_IF
		
	6: 	IF THIS^.xGetTestInfo THEN
            THIS^.sTestCaseName := 'Step 7: ';
            THIS^.sTestCaseCategories := 'General';
            THIS^.diTestCaseTimeout := 3000;
			xDone := TRUE;
		ELSE
			(*TEST SOMETHING HERE*)
			IF (*CONNDITION*) FALSE THEN
				 xDone := TRUE;
			ELSE
				THIS^.sError := '';
				xError := TRUE;
				eError := UnitTestErrors.Failure;
            	eFailureMode := TM.FAILUREMODE.AbortTestCase;
                iError := 1;
			END_IF
        END_IF
    ELSE
        IF THIS^.diTestCaseIndex < 0 THEN
            THIS^.diTestCaseCount := 7;
            xDone := TRUE;
        ELSE
            THIS^.sInfo := 'Invalid test case index';
            eError := UnitTestErrors.Failure;
			xError := TRUE;
        END_IF
END_CASE
END_METHOD

{attribute 'hide'}
METHOD prvResetOutputs : BOOL
SUPER^.prvResetOutputs();

sTestCaseName := '';
sTestCaseCategories := '';
diTestCaseCount := 0;
diTestCaseTimeout := 0;
sInfo := '';
sError := '';
eFailureMode := TM.FAILUREMODE.AbortTestCase;
END_METHOD

{attribute 'hide'}
METHOD prvStart : BOOL
END_METHOD

END_FUNCTION_BLOCK

// Testing/FB_PrinterSerial
FUNCTION_BLOCK FB_PrinterSerial
VAR_INPUT
	sendSampleLabel : BOOL;
	sendClearLabel : BOOL;
	xExecute : BOOL;
END_VAR
VAR_OUTPUT
	xDone : BOOL;(* True, when the test was done succesfully *)
END_VAR
VAR
	iState : INT;
	

	
	(* Settings to communicate with the COM Port *)
	aCom1Params : ARRAY [1..7] OF COM.PARAMETER; 
	aCom2Params : ARRAY [1..7] OF COM.PARAMETER;
	
	como1 : COM.Open;
	comc1 : COM.Close;
	comw1 : COM.Write;

	
	sWrite : STRING := 'Test String!';
	sRead : STRING(25);
	szRead : CAA.SIZE;
	
	xCom1OpenError : BOOL;
	xCom1CloseError : BOOL;
	xCom1WriteError : BOOL;
	executeONS : Standard.R_TRIG;
	sendLabelNow : BOOL;
END_VAR

